// TIA Portal V20 program export: 2 tag tables, 2 data types, 5 data blocks, 11 code blocks (in call order from the OBs), 10 instance data blocks

VAR_GLOBAL   // PLC tag table "PLC_Centralizer_PLC_Production_And_Rework"
   In AT %I500.0 : "IO_Device_Inputs";
   Out AT %Q500.0 : "IO_Device_Outputs";
END_VAR

VAR_GLOBAL   // PLC tag table "PLC_Production_And_Rework"
   Emergency_Stop_Release AT %I0.0 : Bool;
   Sensor_Water_Fountain_Before_Entrace_Functional_Test_Spinner_Conveyor_Belt AT %I0.1 : Bool;
   Sensor_Water_Fountain_Entrace_Functional_Test_Spinner_Conveyor_Belt AT %I0.2 : Bool;
   Sensor_Water_Fountain_Entrace_Functional_Test_After_Spinner_Conveyor_Belt AT %I0.3 : Bool;
   Trigger_Read_Serial_Number_Entrace_Functional_Test AT %I0.4 : Bool;
   Sensor_Water_Fountain_Geting_Exit_Rework_Conveyor_Belt AT %I0.5 : Bool;
   Button_Water_Fountain_Get_Exit_Rework_Conveyor_Belt AT %I0.6 : Bool;
   Trigger_Read_Serial_Number_Exit_Functional_Test AT %I0.7 : Bool;
   Sensor_Water_Fountain_Exit_Functional_Test_Spinner_Conveyor_Belt AT %I1.0 : Bool;
   Sensor_Water_Fountain_Exit_Functional_Test_After_Spinner_Conveyor_Belt AT %I1.1 : Bool;
   Sensor_Water_Fountain_Geting_Entrace_Rework_Conveyor_Belt_Start AT %I1.2 : Bool;
   Sensor_Water_Fountain_Geting_Entrace_Rework_Conveyor_Belt_Finish AT %I1.3 : Bool;
   Carousel_Frequency_Inverter_Fail AT %I1.4 : Bool;
   Conveyor_Belt_Functional_Test_Inverter_Fail AT %I1.5 : Bool;
   Selected_Voltage_220V AT %I8.0 : Bool;
   Selected_Voltage_127V AT %I8.1 : Bool;
   Sensor_Spinner_Entrace_Functional_Test_Position_Withdrawn AT %I8.2 : Bool;
   Sensor_Spinner_Entrace_Functional_Test_Position_Advanced AT %I8.3 : Bool;
   Sensor_Spinner_Exit_Functional_Test_Position_Withdrawn AT %I8.4 : Bool;
   Sensor_Spinner_Exit_Functional_Test_Position_Advanced AT %I8.5 : Bool;
   Digital_Input_20 AT %I8.6 : Bool;
   Digital_Input_21 AT %I8.7 : Bool;
   Digital_Input_22 AT %I9.0 : Bool;
   Digital_Input_23 AT %I9.1 : Bool;
   Digital_Input_24 AT %I9.2 : Bool;
   Digital_Input_25 AT %I9.3 : Bool;
   Digital_Input_26 AT %I9.4 : Bool;
   Digital_Input_27 AT %I9.5 : Bool;
   Digital_Input_28 AT %I9.6 : Bool;
   Digital_Input_29 AT %I9.7 : Bool;
   Analogic_Input_0 AT %IW64 : Int;
   Analogic_Input_1 AT %IW66 : Int;
   Spin_Carousel_Frequency_Inverter_Speed_1 AT %Q0.0 : Bool;
   Spin_Carousel_Frequency_Inverter_Speed_2 AT %Q0.1 : Bool;
   Spin_Carousel_Frequency_Inverter_Speed_3 AT %Q0.2 : Bool;
   Conveyor_Belt_Frequency_Inverter_Speed_1 AT %Q0.3 : Bool;
   Conveyor_Belt_Frequency_Inverter_Speed_2 AT %Q0.4 : Bool;
   Conveyor_Belt_Frequency_Inverter_Speed_3 AT %Q0.5 : Bool;
   Turn_On_Conveyor_Belt_Motor_Spinner_Get_Entrace_Function_Test AT %Q0.6 : Bool;
   Turn_On_Conveyor_Belt_Motor_Rework_Conveyor_Belt_Get_Entrace_Functional_Test AT %Q0.7 : Bool;
   Turn_On_Conveyor_Belt_Motor_Spinner_Get_Exit_Functional_Test AT %Q1.0 : Bool;
   Turn_On_Conveyor_Belt_Motor_Rework_Conveyor_Belt_Get_Exit_Funcional_Test AT %Q1.1 : Bool;
   Open_Air_Pressure AT %Q8.0 : Bool;
   Valve_Advance_Spinner_Entrace_Functional_Test AT %Q8.1 : Bool;
   Valve_Advance_Spinner_Exit_Functional_Test AT %Q8.2 : Bool;
   Signal_Pre_Functional_Test_Production_Line AT %Q8.3 : Bool;
   Digital_Output_14 AT %Q8.4 : Bool;
   Digital_Output_15 AT %Q8.5 : Bool;
   Digital_Output_16 AT %Q8.6 : Bool;
   Digital_Output_17 AT %Q8.7 : Bool;
   Digital_Output_18 AT %Q9.0 : Bool;
   Digital_Output_19 AT %Q9.1 : Bool;
   Digital_Output_20 AT %Q9.2 : Bool;
   Digital_Output_21 AT %Q9.3 : Bool;
   Digital_Output_22 AT %Q9.4 : Bool;
   Digital_Output_23 AT %Q9.5 : Bool;
   Voltage_220V_Selected AT %Q9.6 : Bool;
   Voltage_127V_Selected AT %Q9.7 : Bool;
   Clock_Byte AT %MB0 : Byte;
   Clock_10Hz AT %M0.0 : Bool;
   Clock_5Hz AT %M0.1 : Bool;
   "Clock_2.5Hz" AT %M0.2 : Bool;
   Clock_2Hz AT %M0.3 : Bool;
   "Clock_1.25Hz" AT %M0.4 : Bool;
   Clock_1Hz AT %M0.5 : Bool;
   "Clock_0.625Hz" AT %M0.6 : Bool;
   "Clock_0.5Hz" AT %M0.7 : Bool;
   System_Byte AT %MB1 : Byte;
   FirstScan AT %M1.0 : Bool;
   DiagStatusUpdate AT %M1.1 : Bool;
   AlwaysTRUE AT %M1.2 : Bool;
   AlwaysFALSE AT %M1.3 : Bool;
END_VAR

TYPE "IO_Device_Inputs"
   STRUCT
      Start : Bool;
      Manual_Turn_On_Motor_Caroussel : Bool;
      Manual_Turn_On_Motor_Conveyor_Belt : Bool;
      Water_Foutain_Fail_Functional_Test : Bool;
      Select_Motor_Speed : SInt;
      Carousel_Voltage_Selection : SInt;
   END_STRUCT;
END_TYPE

TYPE "IO_Device_Outputs"
   STRUCT
      Life_Trigger : Bool;
      Emergency_Stop_Release : Bool;
      Trigger_Read_Serial_Number_Entrace_Functional_Test : Bool;
      Trigger_Read_Serial_Number_Exit_Functional_Test : Bool;
      Selected_Voltage_220V : Bool;
      Selected_Voltage_127V : Bool;
      Carousel_Frequency_Inverter_Fail : Bool;
      Conveyor_Belt_Functional_Test_Inverter_Fail : Bool;
   END_STRUCT;
END_TYPE

DATA_BLOCK "DB_Analogic_Input"   // DB2
{ S7_Optimized_Access := 'TRUE' }
// stored: MemoryReserve 100
   VAR
      Real_Analogic_Input_0 : Real;
      Real_Analogic_Input_1 : Real;
      UInt_Analogic_Input_0 : UInt;
      UInt_Analogic_Input_1 : UInt;
   END_VAR
BEGIN
END_DATA_BLOCK

DATA_BLOCK "DB_Contron_Coveyor_Belt"   // DB5
{ S7_Optimized_Access := 'TRUE' }
// stored: MemoryReserve 100
   VAR
      Pause_Conveyor_Belt_And_Carousel_Functional_Test : Bool;
   END_VAR
BEGIN
END_DATA_BLOCK

DATA_BLOCK "DB_Digital_Input"   // DB1
{ S7_Optimized_Access := 'TRUE' }
// stored: MemoryReserve 100
   VAR
      Emergency_Stop_Release : Bool;
      Sensor_Water_Fountain_Before_Entrace_Functional_Test_Spinner_Conveyor_Belt : Bool;
      Sensor_Water_Fountain_Entrace_Functional_Test_Spinner_Conveyor_Belt : Bool;
      Sensor_Water_Fountain_Entrace_Functional_Test_After_Spinner_Conveyor_Belt : Bool;
      Trigger_Read_Serial_Number_Entrace_Functional_Test : Bool;
      Sensor_Water_Fountain_Geting_Exit_Rework_Conveyor_Belt : Bool;
      Button_Water_Fountain_Get_Exit_Rework_Conveyor_Belt : Bool;
      Trigger_Read_Serial_Number_Exit_Functional_Test : Bool;
      Sensor_Water_Fountain_Exit_Functional_Test_Spinner_Conveyor_Belt : Bool;
      Sensor_Water_Fountain_Exit_Functional_Test_After_Spinner_Conveyor_Belt : Bool;
      Sensor_Water_Fountain_Geting_Entrace_Rework_Conveyor_Belt_Start : Bool;
      Sensor_Water_Fountain_Geting_Entrace_Rework_Conveyor_Belt_Finish : Bool;
      Carousel_Frequency_Inverter_Fail : Bool;
      Conveyor_Belt_Functional_Test_Inverter_Fail : Bool;
      Selected_Voltage_220V : Bool;
      Selected_Voltage_127V : Bool;
      Sensor_Spinner_Entrace_Functional_Test_Position_Withdrawn : Bool;
      Sensor_Spinner_Entrace_Functional_Test_Position_Advanced : Bool;
      Sensor_Spinner_Exit_Functional_Test_Position_Withdrawn : Bool;
      Sensor_Spinner_Exit_Functional_Test_Position_Advanced : Bool;
      Digital_Input_20 : Bool;
      Digital_Input_21 : Bool;
      Digital_Input_22 : Bool;
      Digital_Input_23 : Bool;
      Digital_Input_24 : Bool;
      Digital_Input_25 : Bool;
      Digital_Input_26 : Bool;
      Digital_Input_27 : Bool;
      Digital_Input_28 : Bool;
      Digital_Input_29 : Bool;
   END_VAR
BEGIN
END_DATA_BLOCK

DATA_BLOCK "DB_Digital_Output"   // DB3
{ S7_Optimized_Access := 'TRUE' }
// stored: AutoNumber false, MemoryReserve 100
   VAR
      Spin_Carousel_Frequency_Inverter_Speed_1 : Bool;
      Spin_Carousel_Frequency_Inverter_Speed_2 : Bool;
      Spin_Carousel_Frequency_Inverter_Speed_3 : Bool;
      Conveyor_Belt_Frequency_Inverter_Speed_1 : Bool;
      Conveyor_Belt_Frequency_Inverter_Speed_2 : Bool;
      Conveyor_Belt_Frequency_Inverter_Speed_3 : Bool;
      Turn_On_Conveyor_Belt_Motor_Spinner_Get_Entrace_Function_Test : Bool;
      Turn_On_Conveyor_Belt_Motor_Rework_Conveyor_Belt_Get_Entrace_Functional_Test : Bool;
      Turn_On_Conveyor_Belt_Motor_Spinner_Get_Exit_Functional_Test : Bool;
      Turn_On_Conveyor_Belt_Motor_Rework_Conveyor_Belt_Get_Exit_Funcional_Test : Bool;
      Open_Air_Pressure : Bool;
      Valve_Advance_Spinner_Entrace_Functional_Test : Bool;
      Valve_Advance_Spinner_Exit_Functional_Test : Bool;
      Signal_Pre_Functional_Test_Production_Line : Bool;
      Digital_Output_14 : Bool;
      Digital_Output_15 : Bool;
      Digital_Output_16 : Bool;
      Digital_Output_17 : Bool;
      Digital_Output_18 : Bool;
      Digital_Output_19 : Bool;
      Digital_Output_20 : Bool;
      Digital_Output_21 : Bool;
      Digital_Output_22 : Bool;
      Digital_Output_23 : Bool;
      Voltage_220V_Selected : Bool;
      Voltage_127V_Selected : Bool;
   END_VAR
BEGIN
END_DATA_BLOCK

DATA_BLOCK "DB_Info_From_PCL_Centralizer"   // DB4
{ S7_Optimized_Access := 'TRUE' }
// stored: MemoryReserve 100
   VAR
      Start : Bool;
      Manual_Turn_On_Motor_Caroussel : Bool;
      Manual_Turn_On_Motor_Conveyor_Belt : Bool;
      Water_Foutain_Fail_Functional_Test : Bool;
      Select_Motor_Speed : SInt;
      Carousel_Voltage_Selection : SInt;
   END_VAR
BEGIN
END_DATA_BLOCK

ORGANIZATION_BLOCK "Main"   // OB1, LAD, ProgramCycle
TITLE = "Main Program Sweep (Cycle)"
{ S7_Optimized_Access := 'TRUE' }
// stored: SetENOAutomatically false
   VAR_INPUT
      Initial_Call : Bool;   // Initial call of this OB
      Remanence : Bool;   // =True, if remanent data are available
   END_VAR
BEGIN

REGION Network 1
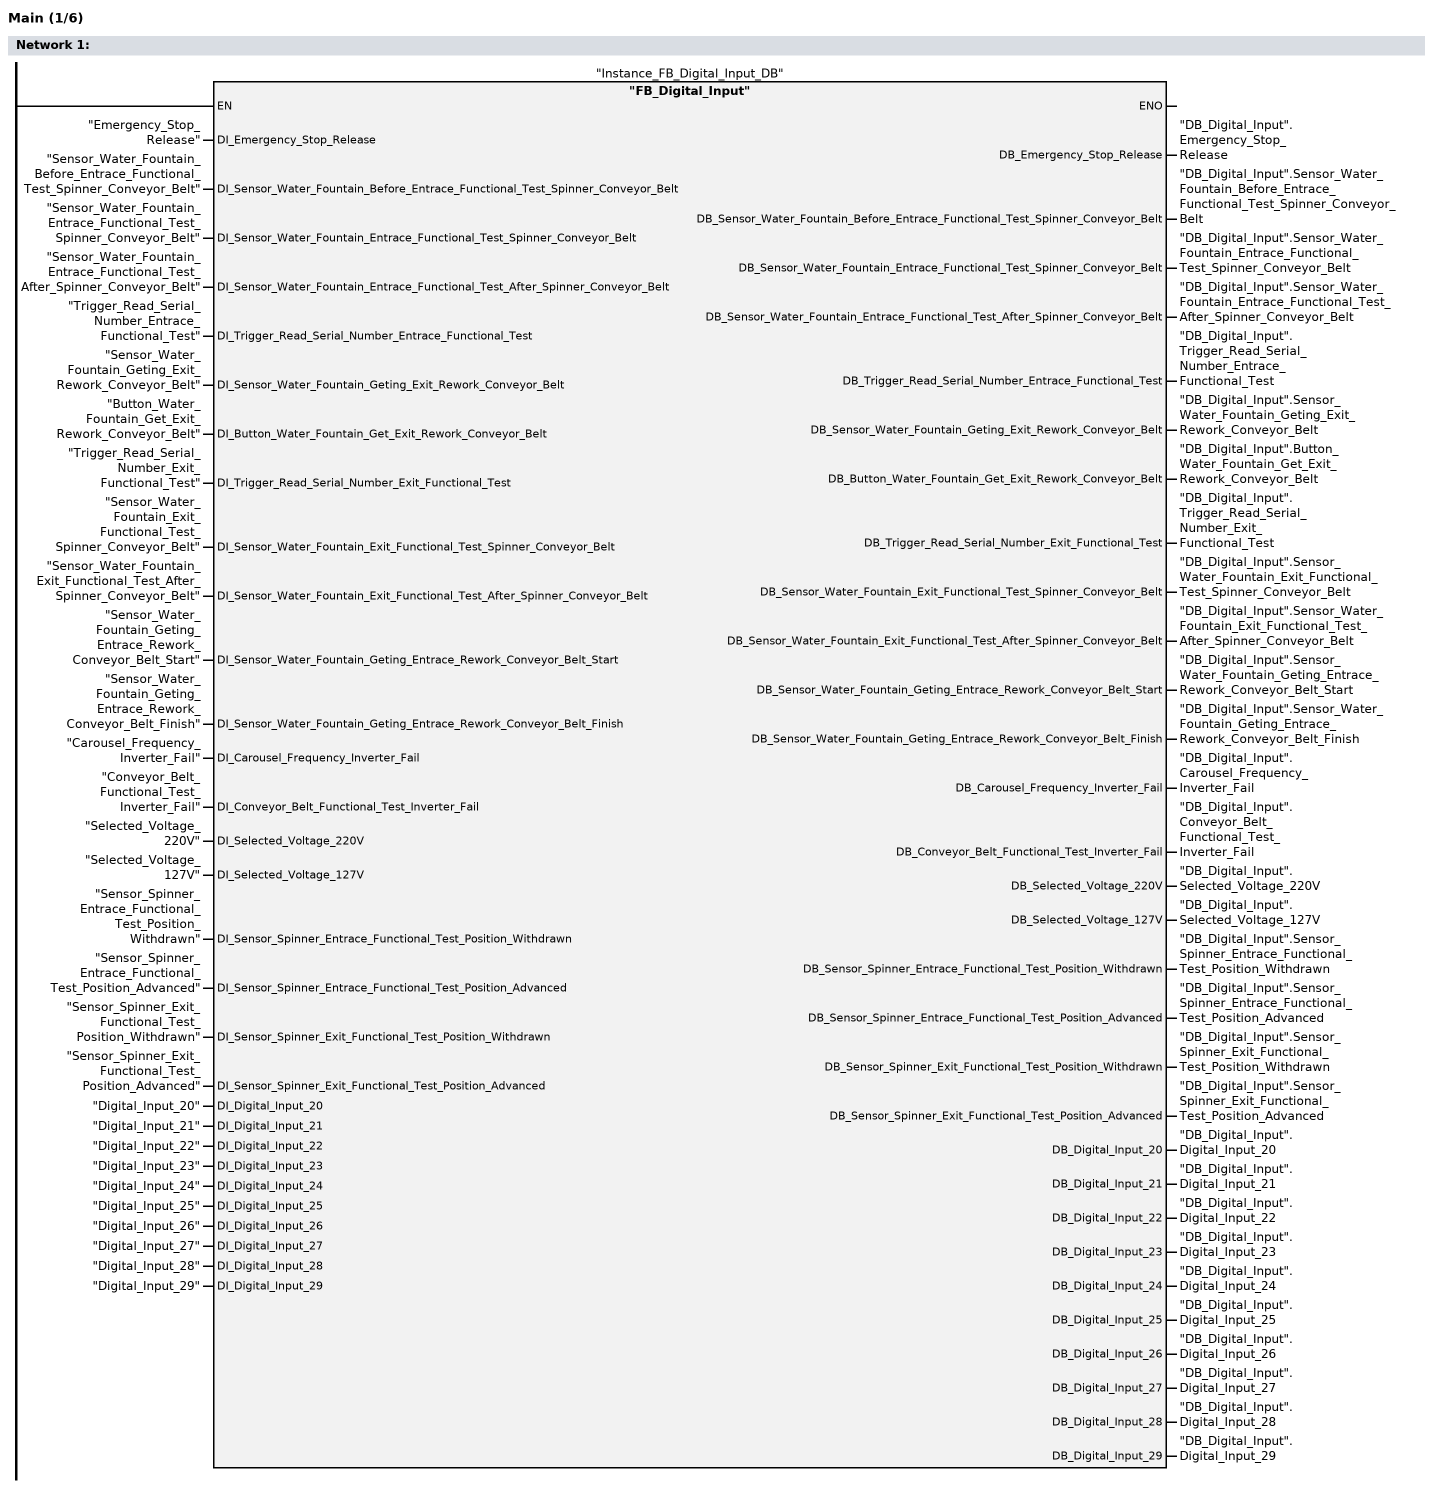
   RUNG wire#powerrail
      "Instance_FB_Digital_Input_DB"(DI_Emergency_Stop_Release := "Emergency_Stop_Release", DI_Sensor_Water_Fountain_Before_Entrace_Functional_Test_Spinner_Conveyor_Belt := "Sensor_Water_Fountain_Before_Entrace_Functional_Test_Spinner_Conveyor_Belt", DI_Sensor_Water_Fountain_Entrace_Functional_Test_Spinner_Conveyor_Belt := "Sensor_Water_Fountain_Entrace_Functional_Test_Spinner_Conveyor_Belt", DI_Sensor_Water_Fountain_Entrace_Functional_Test_After_Spinner_Conveyor_Belt := "Sensor_Water_Fountain_Entrace_Functional_Test_After_Spinner_Conveyor_Belt", DI_Trigger_Read_Serial_Number_Entrace_Functional_Test := "Trigger_Read_Serial_Number_Entrace_Functional_Test", DI_Sensor_Water_Fountain_Geting_Exit_Rework_Conveyor_Belt := "Sensor_Water_Fountain_Geting_Exit_Rework_Conveyor_Belt", DI_Button_Water_Fountain_Get_Exit_Rework_Conveyor_Belt := "Button_Water_Fountain_Get_Exit_Rework_Conveyor_Belt", DI_Trigger_Read_Serial_Number_Exit_Functional_Test := "Trigger_Read_Serial_Number_Exit_Functional_Test", DI_Sensor_Water_Fountain_Exit_Functional_Test_Spinner_Conveyor_Belt := "Sensor_Water_Fountain_Exit_Functional_Test_Spinner_Conveyor_Belt", DI_Sensor_Water_Fountain_Exit_Functional_Test_After_Spinner_Conveyor_Belt := "Sensor_Water_Fountain_Exit_Functional_Test_After_Spinner_Conveyor_Belt", DI_Sensor_Water_Fountain_Geting_Entrace_Rework_Conveyor_Belt_Start := "Sensor_Water_Fountain_Geting_Entrace_Rework_Conveyor_Belt_Start", DI_Sensor_Water_Fountain_Geting_Entrace_Rework_Conveyor_Belt_Finish := "Sensor_Water_Fountain_Geting_Entrace_Rework_Conveyor_Belt_Finish", DI_Carousel_Frequency_Inverter_Fail := "Carousel_Frequency_Inverter_Fail", DI_Conveyor_Belt_Functional_Test_Inverter_Fail := "Conveyor_Belt_Functional_Test_Inverter_Fail", DI_Selected_Voltage_220V := "Selected_Voltage_220V", DI_Selected_Voltage_127V := "Selected_Voltage_127V", DI_Sensor_Spinner_Entrace_Functional_Test_Position_Withdrawn := "Sensor_Spinner_Entrace_Functional_Test_Position_Withdrawn", DI_Sensor_Spinner_Entrace_Functional_Test_Position_Advanced := "Sensor_Spinner_Entrace_Functional_Test_Position_Advanced", DI_Sensor_Spinner_Exit_Functional_Test_Position_Withdrawn := "Sensor_Spinner_Exit_Functional_Test_Position_Withdrawn", DI_Sensor_Spinner_Exit_Functional_Test_Position_Advanced := "Sensor_Spinner_Exit_Functional_Test_Position_Advanced", DI_Digital_Input_20 := "Digital_Input_20", DI_Digital_Input_21 := "Digital_Input_21", DI_Digital_Input_22 := "Digital_Input_22", DI_Digital_Input_23 := "Digital_Input_23", DI_Digital_Input_24 := "Digital_Input_24", DI_Digital_Input_25 := "Digital_Input_25", DI_Digital_Input_26 := "Digital_Input_26", DI_Digital_Input_27 := "Digital_Input_27", DI_Digital_Input_28 := "Digital_Input_28", DI_Digital_Input_29 := "Digital_Input_29", DB_Emergency_Stop_Release => "DB_Digital_Input".Emergency_Stop_Release, DB_Sensor_Water_Fountain_Before_Entrace_Functional_Test_Spinner_Conveyor_Belt => "DB_Digital_Input".Sensor_Water_Fountain_Before_Entrace_Functional_Test_Spinner_Conveyor_Belt, DB_Sensor_Water_Fountain_Entrace_Functional_Test_Spinner_Conveyor_Belt => "DB_Digital_Input".Sensor_Water_Fountain_Entrace_Functional_Test_Spinner_Conveyor_Belt, DB_Sensor_Water_Fountain_Entrace_Functional_Test_After_Spinner_Conveyor_Belt => "DB_Digital_Input".Sensor_Water_Fountain_Entrace_Functional_Test_After_Spinner_Conveyor_Belt, DB_Trigger_Read_Serial_Number_Entrace_Functional_Test => "DB_Digital_Input".Trigger_Read_Serial_Number_Entrace_Functional_Test, DB_Sensor_Water_Fountain_Geting_Exit_Rework_Conveyor_Belt => "DB_Digital_Input".Sensor_Water_Fountain_Geting_Exit_Rework_Conveyor_Belt, DB_Button_Water_Fountain_Get_Exit_Rework_Conveyor_Belt => "DB_Digital_Input".Button_Water_Fountain_Get_Exit_Rework_Conveyor_Belt, DB_Trigger_Read_Serial_Number_Exit_Functional_Test => "DB_Digital_Input".Trigger_Read_Serial_Number_Exit_Functional_Test, DB_Sensor_Water_Fountain_Exit_Functional_Test_Spinner_Conveyor_Belt => "DB_Digital_Input".Sensor_Water_Fountain_Exit_Functional_Test_Spinner_Conveyor_Belt, DB_Sensor_Water_Fountain_Exit_Functional_Test_After_Spinner_Conveyor_Belt => "DB_Digital_Input".Sensor_Water_Fountain_Exit_Functional_Test_After_Spinner_Conveyor_Belt, DB_Sensor_Water_Fountain_Geting_Entrace_Rework_Conveyor_Belt_Start => "DB_Digital_Input".Sensor_Water_Fountain_Geting_Entrace_Rework_Conveyor_Belt_Start, DB_Sensor_Water_Fountain_Geting_Entrace_Rework_Conveyor_Belt_Finish => "DB_Digital_Input".Sensor_Water_Fountain_Geting_Entrace_Rework_Conveyor_Belt_Finish, DB_Carousel_Frequency_Inverter_Fail => "DB_Digital_Input".Carousel_Frequency_Inverter_Fail, DB_Conveyor_Belt_Functional_Test_Inverter_Fail => "DB_Digital_Input".Conveyor_Belt_Functional_Test_Inverter_Fail, DB_Selected_Voltage_220V => "DB_Digital_Input".Selected_Voltage_220V, DB_Selected_Voltage_127V => "DB_Digital_Input".Selected_Voltage_127V, DB_Sensor_Spinner_Entrace_Functional_Test_Position_Withdrawn => "DB_Digital_Input".Sensor_Spinner_Entrace_Functional_Test_Position_Withdrawn, DB_Sensor_Spinner_Entrace_Functional_Test_Position_Advanced => "DB_Digital_Input".Sensor_Spinner_Entrace_Functional_Test_Position_Advanced, DB_Sensor_Spinner_Exit_Functional_Test_Position_Withdrawn => "DB_Digital_Input".Sensor_Spinner_Exit_Functional_Test_Position_Withdrawn, DB_Sensor_Spinner_Exit_Functional_Test_Position_Advanced => "DB_Digital_Input".Sensor_Spinner_Exit_Functional_Test_Position_Advanced, DB_Digital_Input_20 => "DB_Digital_Input".Digital_Input_20, DB_Digital_Input_21 => "DB_Digital_Input".Digital_Input_21, DB_Digital_Input_22 => "DB_Digital_Input".Digital_Input_22, DB_Digital_Input_23 => "DB_Digital_Input".Digital_Input_23, DB_Digital_Input_24 => "DB_Digital_Input".Digital_Input_24, DB_Digital_Input_25 => "DB_Digital_Input".Digital_Input_25, DB_Digital_Input_26 => "DB_Digital_Input".Digital_Input_26, DB_Digital_Input_27 => "DB_Digital_Input".Digital_Input_27, DB_Digital_Input_28 => "DB_Digital_Input".Digital_Input_28, DB_Digital_Input_29 => "DB_Digital_Input".Digital_Input_29)
   END_RUNG
   // the same network as SCL:
   "Instance_FB_Digital_Input_DB"(DI_Emergency_Stop_Release := "Emergency_Stop_Release",   // "FB_Digital_Input"
                           DI_Sensor_Water_Fountain_Before_Entrace_Functional_Test_Spinner_Conveyor_Belt := "Sensor_Water_Fountain_Before_Entrace_Functional_Test_Spinner_Conveyor_Belt",
                           DI_Sensor_Water_Fountain_Entrace_Functional_Test_Spinner_Conveyor_Belt := "Sensor_Water_Fountain_Entrace_Functional_Test_Spinner_Conveyor_Belt",
                           DI_Sensor_Water_Fountain_Entrace_Functional_Test_After_Spinner_Conveyor_Belt := "Sensor_Water_Fountain_Entrace_Functional_Test_After_Spinner_Conveyor_Belt",
                           DI_Trigger_Read_Serial_Number_Entrace_Functional_Test := "Trigger_Read_Serial_Number_Entrace_Functional_Test",
                           DI_Sensor_Water_Fountain_Geting_Exit_Rework_Conveyor_Belt := "Sensor_Water_Fountain_Geting_Exit_Rework_Conveyor_Belt",
                           DI_Button_Water_Fountain_Get_Exit_Rework_Conveyor_Belt := "Button_Water_Fountain_Get_Exit_Rework_Conveyor_Belt",
                           DI_Trigger_Read_Serial_Number_Exit_Functional_Test := "Trigger_Read_Serial_Number_Exit_Functional_Test",
                           DI_Sensor_Water_Fountain_Exit_Functional_Test_Spinner_Conveyor_Belt := "Sensor_Water_Fountain_Exit_Functional_Test_Spinner_Conveyor_Belt",
                           DI_Sensor_Water_Fountain_Exit_Functional_Test_After_Spinner_Conveyor_Belt := "Sensor_Water_Fountain_Exit_Functional_Test_After_Spinner_Conveyor_Belt",
                           DI_Sensor_Water_Fountain_Geting_Entrace_Rework_Conveyor_Belt_Start := "Sensor_Water_Fountain_Geting_Entrace_Rework_Conveyor_Belt_Start",
                           DI_Sensor_Water_Fountain_Geting_Entrace_Rework_Conveyor_Belt_Finish := "Sensor_Water_Fountain_Geting_Entrace_Rework_Conveyor_Belt_Finish",
                           DI_Carousel_Frequency_Inverter_Fail := "Carousel_Frequency_Inverter_Fail",
                           DI_Conveyor_Belt_Functional_Test_Inverter_Fail := "Conveyor_Belt_Functional_Test_Inverter_Fail",
                           DI_Selected_Voltage_220V := "Selected_Voltage_220V",
                           DI_Selected_Voltage_127V := "Selected_Voltage_127V",
                           DI_Sensor_Spinner_Entrace_Functional_Test_Position_Withdrawn := "Sensor_Spinner_Entrace_Functional_Test_Position_Withdrawn",
                           DI_Sensor_Spinner_Entrace_Functional_Test_Position_Advanced := "Sensor_Spinner_Entrace_Functional_Test_Position_Advanced",
                           DI_Sensor_Spinner_Exit_Functional_Test_Position_Withdrawn := "Sensor_Spinner_Exit_Functional_Test_Position_Withdrawn",
                           DI_Sensor_Spinner_Exit_Functional_Test_Position_Advanced := "Sensor_Spinner_Exit_Functional_Test_Position_Advanced",
                           DI_Digital_Input_20 := "Digital_Input_20",
                           DI_Digital_Input_21 := "Digital_Input_21",
                           DI_Digital_Input_22 := "Digital_Input_22",
                           DI_Digital_Input_23 := "Digital_Input_23",
                           DI_Digital_Input_24 := "Digital_Input_24",
                           DI_Digital_Input_25 := "Digital_Input_25",
                           DI_Digital_Input_26 := "Digital_Input_26",
                           DI_Digital_Input_27 := "Digital_Input_27",
                           DI_Digital_Input_28 := "Digital_Input_28",
                           DI_Digital_Input_29 := "Digital_Input_29",
                           DB_Emergency_Stop_Release => "DB_Digital_Input".Emergency_Stop_Release,
                           DB_Sensor_Water_Fountain_Before_Entrace_Functional_Test_Spinner_Conveyor_Belt => "DB_Digital_Input".Sensor_Water_Fountain_Before_Entrace_Functional_Test_Spinner_Conveyor_Belt,
                           DB_Sensor_Water_Fountain_Entrace_Functional_Test_Spinner_Conveyor_Belt => "DB_Digital_Input".Sensor_Water_Fountain_Entrace_Functional_Test_Spinner_Conveyor_Belt,
                           DB_Sensor_Water_Fountain_Entrace_Functional_Test_After_Spinner_Conveyor_Belt => "DB_Digital_Input".Sensor_Water_Fountain_Entrace_Functional_Test_After_Spinner_Conveyor_Belt,
                           DB_Trigger_Read_Serial_Number_Entrace_Functional_Test => "DB_Digital_Input".Trigger_Read_Serial_Number_Entrace_Functional_Test,
                           DB_Sensor_Water_Fountain_Geting_Exit_Rework_Conveyor_Belt => "DB_Digital_Input".Sensor_Water_Fountain_Geting_Exit_Rework_Conveyor_Belt,
                           DB_Button_Water_Fountain_Get_Exit_Rework_Conveyor_Belt => "DB_Digital_Input".Button_Water_Fountain_Get_Exit_Rework_Conveyor_Belt,
                           DB_Trigger_Read_Serial_Number_Exit_Functional_Test => "DB_Digital_Input".Trigger_Read_Serial_Number_Exit_Functional_Test,
                           DB_Sensor_Water_Fountain_Exit_Functional_Test_Spinner_Conveyor_Belt => "DB_Digital_Input".Sensor_Water_Fountain_Exit_Functional_Test_Spinner_Conveyor_Belt,
                           DB_Sensor_Water_Fountain_Exit_Functional_Test_After_Spinner_Conveyor_Belt => "DB_Digital_Input".Sensor_Water_Fountain_Exit_Functional_Test_After_Spinner_Conveyor_Belt,
                           DB_Sensor_Water_Fountain_Geting_Entrace_Rework_Conveyor_Belt_Start => "DB_Digital_Input".Sensor_Water_Fountain_Geting_Entrace_Rework_Conveyor_Belt_Start,
                           DB_Sensor_Water_Fountain_Geting_Entrace_Rework_Conveyor_Belt_Finish => "DB_Digital_Input".Sensor_Water_Fountain_Geting_Entrace_Rework_Conveyor_Belt_Finish,
                           DB_Carousel_Frequency_Inverter_Fail => "DB_Digital_Input".Carousel_Frequency_Inverter_Fail,
                           DB_Conveyor_Belt_Functional_Test_Inverter_Fail => "DB_Digital_Input".Conveyor_Belt_Functional_Test_Inverter_Fail,
                           DB_Selected_Voltage_220V => "DB_Digital_Input".Selected_Voltage_220V,
                           DB_Selected_Voltage_127V => "DB_Digital_Input".Selected_Voltage_127V,
                           DB_Sensor_Spinner_Entrace_Functional_Test_Position_Withdrawn => "DB_Digital_Input".Sensor_Spinner_Entrace_Functional_Test_Position_Withdrawn,
                           DB_Sensor_Spinner_Entrace_Functional_Test_Position_Advanced => "DB_Digital_Input".Sensor_Spinner_Entrace_Functional_Test_Position_Advanced,
                           DB_Sensor_Spinner_Exit_Functional_Test_Position_Withdrawn => "DB_Digital_Input".Sensor_Spinner_Exit_Functional_Test_Position_Withdrawn,
                           DB_Sensor_Spinner_Exit_Functional_Test_Position_Advanced => "DB_Digital_Input".Sensor_Spinner_Exit_Functional_Test_Position_Advanced,
                           DB_Digital_Input_20 => "DB_Digital_Input".Digital_Input_20,
                           DB_Digital_Input_21 => "DB_Digital_Input".Digital_Input_21,
                           DB_Digital_Input_22 => "DB_Digital_Input".Digital_Input_22,
                           DB_Digital_Input_23 => "DB_Digital_Input".Digital_Input_23,
                           DB_Digital_Input_24 => "DB_Digital_Input".Digital_Input_24,
                           DB_Digital_Input_25 => "DB_Digital_Input".Digital_Input_25,
                           DB_Digital_Input_26 => "DB_Digital_Input".Digital_Input_26,
                           DB_Digital_Input_27 => "DB_Digital_Input".Digital_Input_27,
                           DB_Digital_Input_28 => "DB_Digital_Input".Digital_Input_28,
                           DB_Digital_Input_29 => "DB_Digital_Input".Digital_Input_29);
END_REGION

REGION Network 2
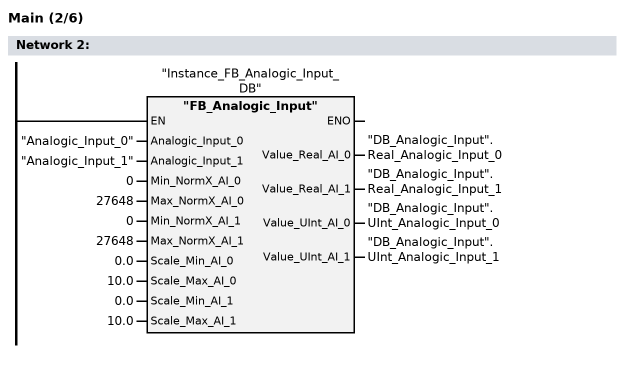
   RUNG wire#powerrail
      "Instance_FB_Analogic_Input_DB"(Analogic_Input_0 := "Analogic_Input_0", Analogic_Input_1 := "Analogic_Input_1", Min_NormX_AI_0 := 0, Max_NormX_AI_0 := 27648, Min_NormX_AI_1 := 0, Max_NormX_AI_1 := 27648, Scale_Min_AI_0 := 0.0, Scale_Max_AI_0 := 10.0, Scale_Min_AI_1 := 0.0, Scale_Max_AI_1 := 10.0, Value_Real_AI_0 => "DB_Analogic_Input".Real_Analogic_Input_0, Value_Real_AI_1 => "DB_Analogic_Input".Real_Analogic_Input_1, Value_UInt_AI_0 => "DB_Analogic_Input".UInt_Analogic_Input_0, Value_UInt_AI_1 => "DB_Analogic_Input".UInt_Analogic_Input_1)
   END_RUNG
   // the same network as SCL:
   "Instance_FB_Analogic_Input_DB"(Analogic_Input_0 := "Analogic_Input_0",   // "FB_Analogic_Input"
                           Analogic_Input_1 := "Analogic_Input_1",
                           Min_NormX_AI_0 := 0,
                           Max_NormX_AI_0 := 27648,
                           Min_NormX_AI_1 := 0,
                           Max_NormX_AI_1 := 27648,
                           Scale_Min_AI_0 := 0.0,
                           Scale_Max_AI_0 := 10.0,
                           Scale_Min_AI_1 := 0.0,
                           Scale_Max_AI_1 := 10.0,
                           Value_Real_AI_0 => "DB_Analogic_Input".Real_Analogic_Input_0,
                           Value_Real_AI_1 => "DB_Analogic_Input".Real_Analogic_Input_1,
                           Value_UInt_AI_0 => "DB_Analogic_Input".UInt_Analogic_Input_0,
                           Value_UInt_AI_1 => "DB_Analogic_Input".UInt_Analogic_Input_1);
END_REGION

REGION Network 3
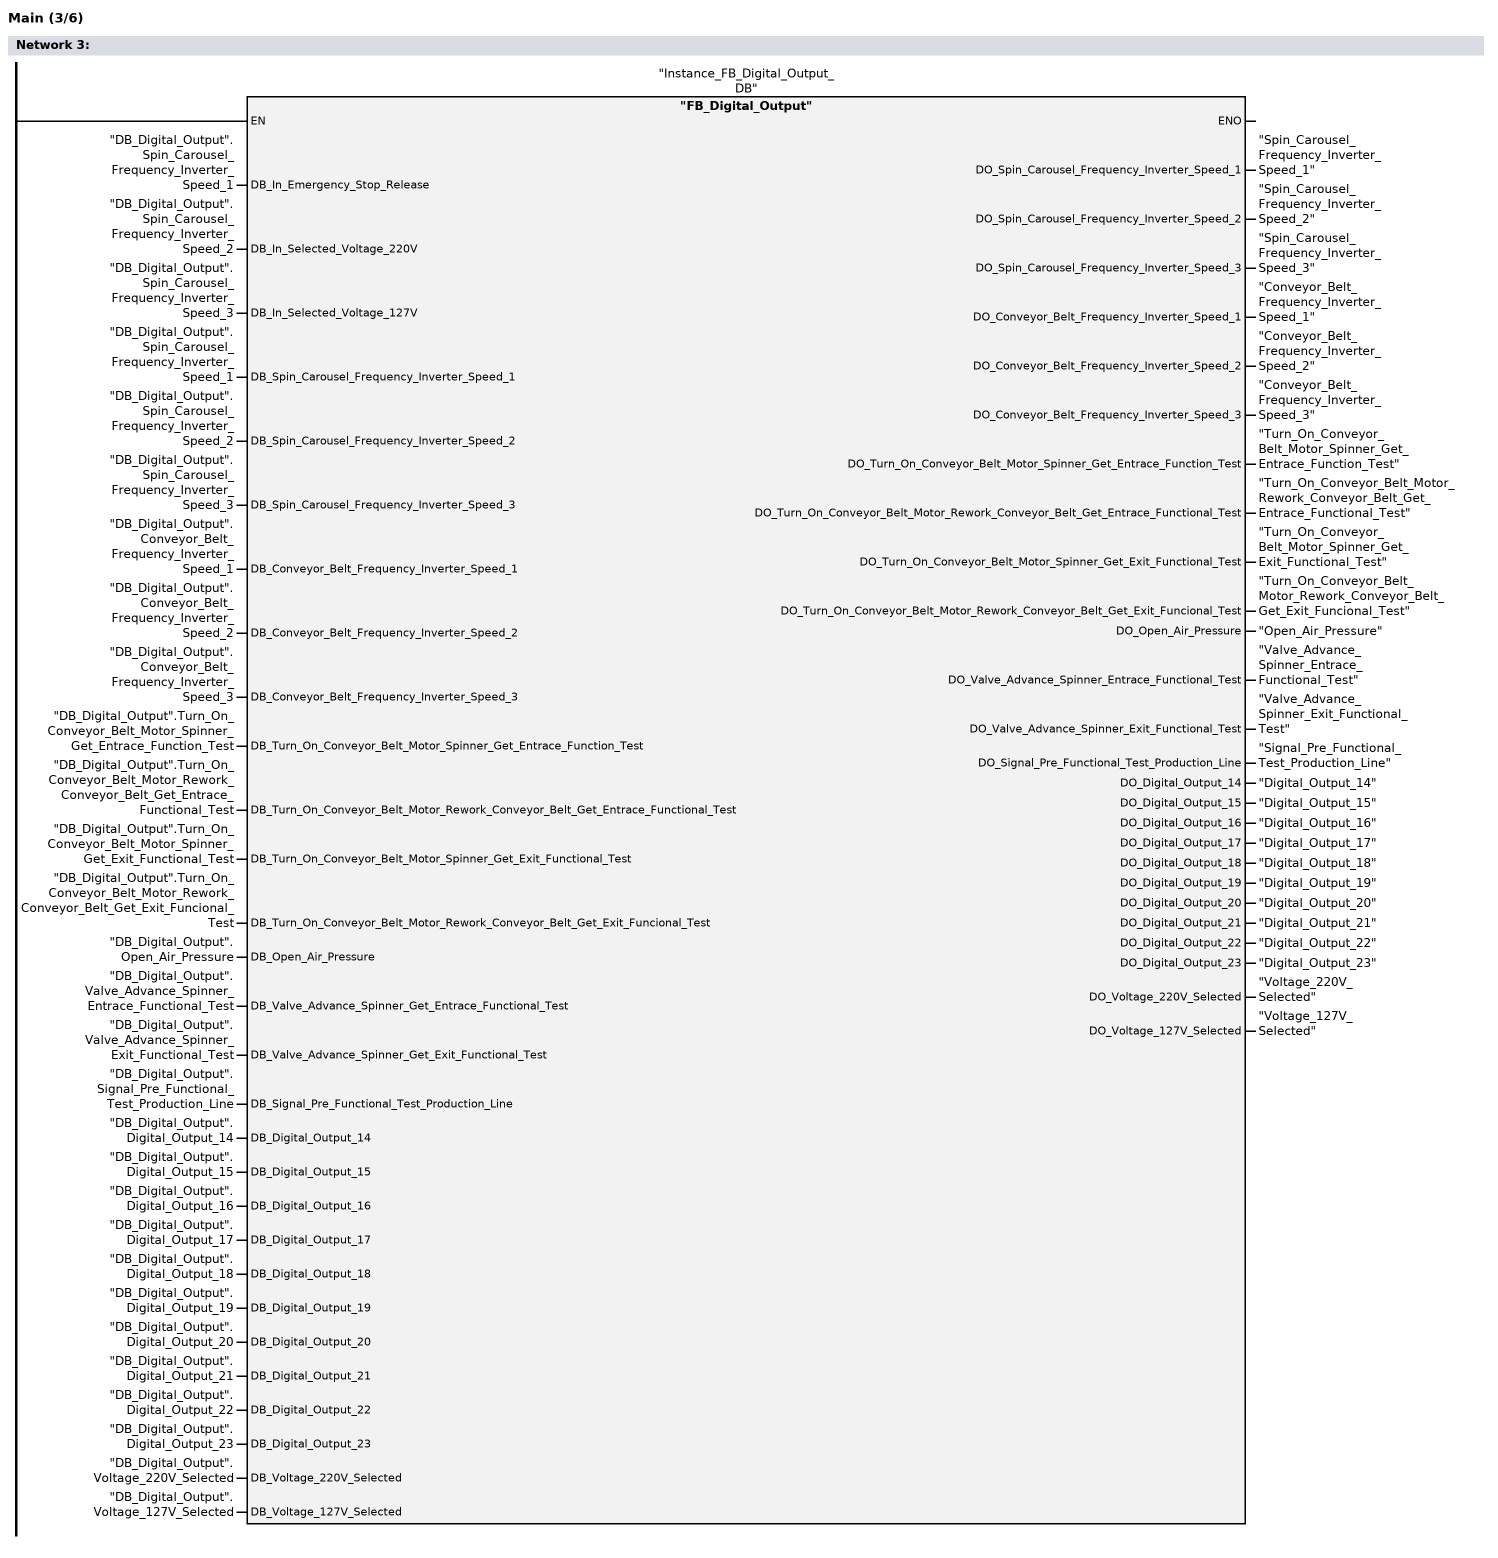
   RUNG wire#powerrail
      "Instance_FB_Digital_Output_DB"(DB_In_Emergency_Stop_Release := "DB_Digital_Output".Spin_Carousel_Frequency_Inverter_Speed_1, DB_In_Selected_Voltage_220V := "DB_Digital_Output".Spin_Carousel_Frequency_Inverter_Speed_2, DB_In_Selected_Voltage_127V := "DB_Digital_Output".Spin_Carousel_Frequency_Inverter_Speed_3, DB_Spin_Carousel_Frequency_Inverter_Speed_1 := "DB_Digital_Output".Spin_Carousel_Frequency_Inverter_Speed_1, DB_Spin_Carousel_Frequency_Inverter_Speed_2 := "DB_Digital_Output".Spin_Carousel_Frequency_Inverter_Speed_2, DB_Spin_Carousel_Frequency_Inverter_Speed_3 := "DB_Digital_Output".Spin_Carousel_Frequency_Inverter_Speed_3, DB_Conveyor_Belt_Frequency_Inverter_Speed_1 := "DB_Digital_Output".Conveyor_Belt_Frequency_Inverter_Speed_1, DB_Conveyor_Belt_Frequency_Inverter_Speed_2 := "DB_Digital_Output".Conveyor_Belt_Frequency_Inverter_Speed_2, DB_Conveyor_Belt_Frequency_Inverter_Speed_3 := "DB_Digital_Output".Conveyor_Belt_Frequency_Inverter_Speed_3, DB_Turn_On_Conveyor_Belt_Motor_Spinner_Get_Entrace_Function_Test := "DB_Digital_Output".Turn_On_Conveyor_Belt_Motor_Spinner_Get_Entrace_Function_Test, DB_Turn_On_Conveyor_Belt_Motor_Rework_Conveyor_Belt_Get_Entrace_Functional_Test := "DB_Digital_Output".Turn_On_Conveyor_Belt_Motor_Rework_Conveyor_Belt_Get_Entrace_Functional_Test, DB_Turn_On_Conveyor_Belt_Motor_Spinner_Get_Exit_Functional_Test := "DB_Digital_Output".Turn_On_Conveyor_Belt_Motor_Spinner_Get_Exit_Functional_Test, DB_Turn_On_Conveyor_Belt_Motor_Rework_Conveyor_Belt_Get_Exit_Funcional_Test := "DB_Digital_Output".Turn_On_Conveyor_Belt_Motor_Rework_Conveyor_Belt_Get_Exit_Funcional_Test, DB_Open_Air_Pressure := "DB_Digital_Output".Open_Air_Pressure, DB_Valve_Advance_Spinner_Get_Entrace_Functional_Test := "DB_Digital_Output".Valve_Advance_Spinner_Entrace_Functional_Test, DB_Valve_Advance_Spinner_Get_Exit_Functional_Test := "DB_Digital_Output".Valve_Advance_Spinner_Exit_Functional_Test, DB_Signal_Pre_Functional_Test_Production_Line := "DB_Digital_Output".Signal_Pre_Functional_Test_Production_Line, DB_Digital_Output_14 := "DB_Digital_Output".Digital_Output_14, DB_Digital_Output_15 := "DB_Digital_Output".Digital_Output_15, DB_Digital_Output_16 := "DB_Digital_Output".Digital_Output_16, DB_Digital_Output_17 := "DB_Digital_Output".Digital_Output_17, DB_Digital_Output_18 := "DB_Digital_Output".Digital_Output_18, DB_Digital_Output_19 := "DB_Digital_Output".Digital_Output_19, DB_Digital_Output_20 := "DB_Digital_Output".Digital_Output_20, DB_Digital_Output_21 := "DB_Digital_Output".Digital_Output_21, DB_Digital_Output_22 := "DB_Digital_Output".Digital_Output_22, DB_Digital_Output_23 := "DB_Digital_Output".Digital_Output_23, DB_Voltage_220V_Selected := "DB_Digital_Output".Voltage_220V_Selected, DB_Voltage_127V_Selected := "DB_Digital_Output".Voltage_127V_Selected, DO_Spin_Carousel_Frequency_Inverter_Speed_1 => "Spin_Carousel_Frequency_Inverter_Speed_1", DO_Spin_Carousel_Frequency_Inverter_Speed_2 => "Spin_Carousel_Frequency_Inverter_Speed_2", DO_Spin_Carousel_Frequency_Inverter_Speed_3 => "Spin_Carousel_Frequency_Inverter_Speed_3", DO_Conveyor_Belt_Frequency_Inverter_Speed_1 => "Conveyor_Belt_Frequency_Inverter_Speed_1", DO_Conveyor_Belt_Frequency_Inverter_Speed_2 => "Conveyor_Belt_Frequency_Inverter_Speed_2", DO_Conveyor_Belt_Frequency_Inverter_Speed_3 => "Conveyor_Belt_Frequency_Inverter_Speed_3", DO_Turn_On_Conveyor_Belt_Motor_Spinner_Get_Entrace_Function_Test => "Turn_On_Conveyor_Belt_Motor_Spinner_Get_Entrace_Function_Test", DO_Turn_On_Conveyor_Belt_Motor_Rework_Conveyor_Belt_Get_Entrace_Functional_Test => "Turn_On_Conveyor_Belt_Motor_Rework_Conveyor_Belt_Get_Entrace_Functional_Test", DO_Turn_On_Conveyor_Belt_Motor_Spinner_Get_Exit_Functional_Test => "Turn_On_Conveyor_Belt_Motor_Spinner_Get_Exit_Functional_Test", DO_Turn_On_Conveyor_Belt_Motor_Rework_Conveyor_Belt_Get_Exit_Funcional_Test => "Turn_On_Conveyor_Belt_Motor_Rework_Conveyor_Belt_Get_Exit_Funcional_Test", DO_Open_Air_Pressure => "Open_Air_Pressure", DO_Valve_Advance_Spinner_Entrace_Functional_Test => "Valve_Advance_Spinner_Entrace_Functional_Test", DO_Valve_Advance_Spinner_Exit_Functional_Test => "Valve_Advance_Spinner_Exit_Functional_Test", DO_Signal_Pre_Functional_Test_Production_Line => "Signal_Pre_Functional_Test_Production_Line", DO_Digital_Output_14 => "Digital_Output_14", DO_Digital_Output_15 => "Digital_Output_15", DO_Digital_Output_16 => "Digital_Output_16", DO_Digital_Output_17 => "Digital_Output_17", DO_Digital_Output_18 => "Digital_Output_18", DO_Digital_Output_19 => "Digital_Output_19", DO_Digital_Output_20 => "Digital_Output_20", DO_Digital_Output_21 => "Digital_Output_21", DO_Digital_Output_22 => "Digital_Output_22", DO_Digital_Output_23 => "Digital_Output_23", DO_Voltage_220V_Selected => "Voltage_220V_Selected", DO_Voltage_127V_Selected => "Voltage_127V_Selected")
   END_RUNG
   // the same network as SCL:
   "Instance_FB_Digital_Output_DB"(DB_In_Emergency_Stop_Release := "DB_Digital_Output".Spin_Carousel_Frequency_Inverter_Speed_1,   // "FB_Digital_Output"
                           DB_In_Selected_Voltage_220V := "DB_Digital_Output".Spin_Carousel_Frequency_Inverter_Speed_2,
                           DB_In_Selected_Voltage_127V := "DB_Digital_Output".Spin_Carousel_Frequency_Inverter_Speed_3,
                           DB_Spin_Carousel_Frequency_Inverter_Speed_1 := "DB_Digital_Output".Spin_Carousel_Frequency_Inverter_Speed_1,
                           DB_Spin_Carousel_Frequency_Inverter_Speed_2 := "DB_Digital_Output".Spin_Carousel_Frequency_Inverter_Speed_2,
                           DB_Spin_Carousel_Frequency_Inverter_Speed_3 := "DB_Digital_Output".Spin_Carousel_Frequency_Inverter_Speed_3,
                           DB_Conveyor_Belt_Frequency_Inverter_Speed_1 := "DB_Digital_Output".Conveyor_Belt_Frequency_Inverter_Speed_1,
                           DB_Conveyor_Belt_Frequency_Inverter_Speed_2 := "DB_Digital_Output".Conveyor_Belt_Frequency_Inverter_Speed_2,
                           DB_Conveyor_Belt_Frequency_Inverter_Speed_3 := "DB_Digital_Output".Conveyor_Belt_Frequency_Inverter_Speed_3,
                           DB_Turn_On_Conveyor_Belt_Motor_Spinner_Get_Entrace_Function_Test := "DB_Digital_Output".Turn_On_Conveyor_Belt_Motor_Spinner_Get_Entrace_Function_Test,
                           DB_Turn_On_Conveyor_Belt_Motor_Rework_Conveyor_Belt_Get_Entrace_Functional_Test := "DB_Digital_Output".Turn_On_Conveyor_Belt_Motor_Rework_Conveyor_Belt_Get_Entrace_Functional_Test,
                           DB_Turn_On_Conveyor_Belt_Motor_Spinner_Get_Exit_Functional_Test := "DB_Digital_Output".Turn_On_Conveyor_Belt_Motor_Spinner_Get_Exit_Functional_Test,
                           DB_Turn_On_Conveyor_Belt_Motor_Rework_Conveyor_Belt_Get_Exit_Funcional_Test := "DB_Digital_Output".Turn_On_Conveyor_Belt_Motor_Rework_Conveyor_Belt_Get_Exit_Funcional_Test,
                           DB_Open_Air_Pressure := "DB_Digital_Output".Open_Air_Pressure,
                           DB_Valve_Advance_Spinner_Get_Entrace_Functional_Test := "DB_Digital_Output".Valve_Advance_Spinner_Entrace_Functional_Test,
                           DB_Valve_Advance_Spinner_Get_Exit_Functional_Test := "DB_Digital_Output".Valve_Advance_Spinner_Exit_Functional_Test,
                           DB_Signal_Pre_Functional_Test_Production_Line := "DB_Digital_Output".Signal_Pre_Functional_Test_Production_Line,
                           DB_Digital_Output_14 := "DB_Digital_Output".Digital_Output_14,
                           DB_Digital_Output_15 := "DB_Digital_Output".Digital_Output_15,
                           DB_Digital_Output_16 := "DB_Digital_Output".Digital_Output_16,
                           DB_Digital_Output_17 := "DB_Digital_Output".Digital_Output_17,
                           DB_Digital_Output_18 := "DB_Digital_Output".Digital_Output_18,
                           DB_Digital_Output_19 := "DB_Digital_Output".Digital_Output_19,
                           DB_Digital_Output_20 := "DB_Digital_Output".Digital_Output_20,
                           DB_Digital_Output_21 := "DB_Digital_Output".Digital_Output_21,
                           DB_Digital_Output_22 := "DB_Digital_Output".Digital_Output_22,
                           DB_Digital_Output_23 := "DB_Digital_Output".Digital_Output_23,
                           DB_Voltage_220V_Selected := "DB_Digital_Output".Voltage_220V_Selected,
                           DB_Voltage_127V_Selected := "DB_Digital_Output".Voltage_127V_Selected,
                           DO_Spin_Carousel_Frequency_Inverter_Speed_1 => "Spin_Carousel_Frequency_Inverter_Speed_1",
                           DO_Spin_Carousel_Frequency_Inverter_Speed_2 => "Spin_Carousel_Frequency_Inverter_Speed_2",
                           DO_Spin_Carousel_Frequency_Inverter_Speed_3 => "Spin_Carousel_Frequency_Inverter_Speed_3",
                           DO_Conveyor_Belt_Frequency_Inverter_Speed_1 => "Conveyor_Belt_Frequency_Inverter_Speed_1",
                           DO_Conveyor_Belt_Frequency_Inverter_Speed_2 => "Conveyor_Belt_Frequency_Inverter_Speed_2",
                           DO_Conveyor_Belt_Frequency_Inverter_Speed_3 => "Conveyor_Belt_Frequency_Inverter_Speed_3",
                           DO_Turn_On_Conveyor_Belt_Motor_Spinner_Get_Entrace_Function_Test => "Turn_On_Conveyor_Belt_Motor_Spinner_Get_Entrace_Function_Test",
                           DO_Turn_On_Conveyor_Belt_Motor_Rework_Conveyor_Belt_Get_Entrace_Functional_Test => "Turn_On_Conveyor_Belt_Motor_Rework_Conveyor_Belt_Get_Entrace_Functional_Test",
                           DO_Turn_On_Conveyor_Belt_Motor_Spinner_Get_Exit_Functional_Test => "Turn_On_Conveyor_Belt_Motor_Spinner_Get_Exit_Functional_Test",
                           DO_Turn_On_Conveyor_Belt_Motor_Rework_Conveyor_Belt_Get_Exit_Funcional_Test => "Turn_On_Conveyor_Belt_Motor_Rework_Conveyor_Belt_Get_Exit_Funcional_Test",
                           DO_Open_Air_Pressure => "Open_Air_Pressure",
                           DO_Valve_Advance_Spinner_Entrace_Functional_Test => "Valve_Advance_Spinner_Entrace_Functional_Test",
                           DO_Valve_Advance_Spinner_Exit_Functional_Test => "Valve_Advance_Spinner_Exit_Functional_Test",
                           DO_Signal_Pre_Functional_Test_Production_Line => "Signal_Pre_Functional_Test_Production_Line",
                           DO_Digital_Output_14 => "Digital_Output_14",
                           DO_Digital_Output_15 => "Digital_Output_15",
                           DO_Digital_Output_16 => "Digital_Output_16",
                           DO_Digital_Output_17 => "Digital_Output_17",
                           DO_Digital_Output_18 => "Digital_Output_18",
                           DO_Digital_Output_19 => "Digital_Output_19",
                           DO_Digital_Output_20 => "Digital_Output_20",
                           DO_Digital_Output_21 => "Digital_Output_21",
                           DO_Digital_Output_22 => "Digital_Output_22",
                           DO_Digital_Output_23 => "Digital_Output_23",
                           DO_Voltage_220V_Selected => "Voltage_220V_Selected",
                           DO_Voltage_127V_Selected => "Voltage_127V_Selected");
END_REGION

REGION Network 4
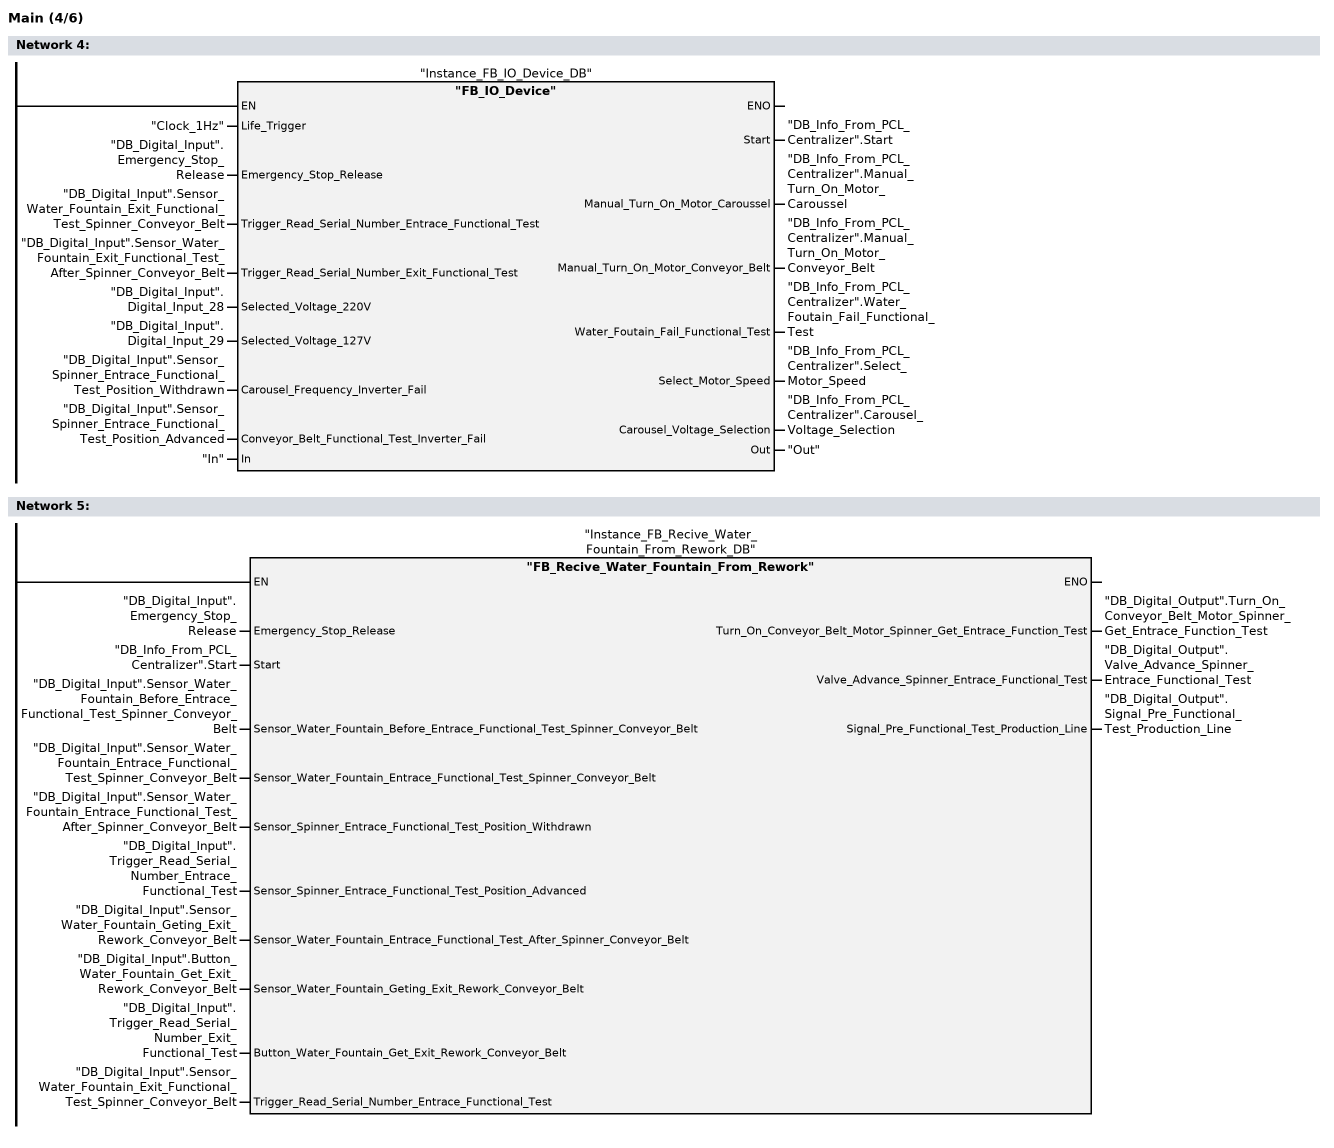
   RUNG wire#powerrail
      "Instance_FB_IO_Device_DB"(Life_Trigger := "Clock_1Hz", Emergency_Stop_Release := "DB_Digital_Input".Emergency_Stop_Release, Trigger_Read_Serial_Number_Entrace_Functional_Test := "DB_Digital_Input".Sensor_Water_Fountain_Exit_Functional_Test_Spinner_Conveyor_Belt, Trigger_Read_Serial_Number_Exit_Functional_Test := "DB_Digital_Input".Sensor_Water_Fountain_Exit_Functional_Test_After_Spinner_Conveyor_Belt, Selected_Voltage_220V := "DB_Digital_Input".Digital_Input_28, Selected_Voltage_127V := "DB_Digital_Input".Digital_Input_29, Carousel_Frequency_Inverter_Fail := "DB_Digital_Input".Sensor_Spinner_Entrace_Functional_Test_Position_Withdrawn, Conveyor_Belt_Functional_Test_Inverter_Fail := "DB_Digital_Input".Sensor_Spinner_Entrace_Functional_Test_Position_Advanced, In := "In", Start => "DB_Info_From_PCL_Centralizer".Start, Manual_Turn_On_Motor_Caroussel => "DB_Info_From_PCL_Centralizer".Manual_Turn_On_Motor_Caroussel, Manual_Turn_On_Motor_Conveyor_Belt => "DB_Info_From_PCL_Centralizer".Manual_Turn_On_Motor_Conveyor_Belt, Water_Foutain_Fail_Functional_Test => "DB_Info_From_PCL_Centralizer".Water_Foutain_Fail_Functional_Test, Select_Motor_Speed => "DB_Info_From_PCL_Centralizer".Select_Motor_Speed, Carousel_Voltage_Selection => "DB_Info_From_PCL_Centralizer".Carousel_Voltage_Selection, Out => "Out")
   END_RUNG
   // the same network as SCL:
   "Instance_FB_IO_Device_DB"(Life_Trigger := "Clock_1Hz",   // "FB_IO_Device"
                           Emergency_Stop_Release := "DB_Digital_Input".Emergency_Stop_Release,
                           Trigger_Read_Serial_Number_Entrace_Functional_Test := "DB_Digital_Input".Sensor_Water_Fountain_Exit_Functional_Test_Spinner_Conveyor_Belt,
                           Trigger_Read_Serial_Number_Exit_Functional_Test := "DB_Digital_Input".Sensor_Water_Fountain_Exit_Functional_Test_After_Spinner_Conveyor_Belt,
                           Selected_Voltage_220V := "DB_Digital_Input".Digital_Input_28,
                           Selected_Voltage_127V := "DB_Digital_Input".Digital_Input_29,
                           Carousel_Frequency_Inverter_Fail := "DB_Digital_Input".Sensor_Spinner_Entrace_Functional_Test_Position_Withdrawn,
                           Conveyor_Belt_Functional_Test_Inverter_Fail := "DB_Digital_Input".Sensor_Spinner_Entrace_Functional_Test_Position_Advanced,
                           In := "In",
                           Start => "DB_Info_From_PCL_Centralizer".Start,
                           Manual_Turn_On_Motor_Caroussel => "DB_Info_From_PCL_Centralizer".Manual_Turn_On_Motor_Caroussel,
                           Manual_Turn_On_Motor_Conveyor_Belt => "DB_Info_From_PCL_Centralizer".Manual_Turn_On_Motor_Conveyor_Belt,
                           Water_Foutain_Fail_Functional_Test => "DB_Info_From_PCL_Centralizer".Water_Foutain_Fail_Functional_Test,
                           Select_Motor_Speed => "DB_Info_From_PCL_Centralizer".Select_Motor_Speed,
                           Carousel_Voltage_Selection => "DB_Info_From_PCL_Centralizer".Carousel_Voltage_Selection,
                           Out => "Out");
END_REGION

REGION Network 5
   RUNG wire#powerrail
      "Instance_FB_Recive_Water_Fountain_From_Rework_DB"(Emergency_Stop_Release := "DB_Digital_Input".Emergency_Stop_Release, Start := "DB_Info_From_PCL_Centralizer".Start, Sensor_Water_Fountain_Before_Entrace_Functional_Test_Spinner_Conveyor_Belt := "DB_Digital_Input".Sensor_Water_Fountain_Before_Entrace_Functional_Test_Spinner_Conveyor_Belt, Sensor_Water_Fountain_Entrace_Functional_Test_Spinner_Conveyor_Belt := "DB_Digital_Input".Sensor_Water_Fountain_Entrace_Functional_Test_Spinner_Conveyor_Belt, Sensor_Spinner_Entrace_Functional_Test_Position_Withdrawn := "DB_Digital_Input".Sensor_Water_Fountain_Entrace_Functional_Test_After_Spinner_Conveyor_Belt, Sensor_Spinner_Entrace_Functional_Test_Position_Advanced := "DB_Digital_Input".Trigger_Read_Serial_Number_Entrace_Functional_Test, Sensor_Water_Fountain_Entrace_Functional_Test_After_Spinner_Conveyor_Belt := "DB_Digital_Input".Sensor_Water_Fountain_Geting_Exit_Rework_Conveyor_Belt, Sensor_Water_Fountain_Geting_Exit_Rework_Conveyor_Belt := "DB_Digital_Input".Button_Water_Fountain_Get_Exit_Rework_Conveyor_Belt, Button_Water_Fountain_Get_Exit_Rework_Conveyor_Belt := "DB_Digital_Input".Trigger_Read_Serial_Number_Exit_Functional_Test, Trigger_Read_Serial_Number_Entrace_Functional_Test := "DB_Digital_Input".Sensor_Water_Fountain_Exit_Functional_Test_Spinner_Conveyor_Belt, Turn_On_Conveyor_Belt_Motor_Spinner_Get_Entrace_Function_Test => "DB_Digital_Output".Turn_On_Conveyor_Belt_Motor_Spinner_Get_Entrace_Function_Test, Valve_Advance_Spinner_Entrace_Functional_Test => "DB_Digital_Output".Valve_Advance_Spinner_Entrace_Functional_Test, Signal_Pre_Functional_Test_Production_Line => "DB_Digital_Output".Signal_Pre_Functional_Test_Production_Line)
   END_RUNG
   // the same network as SCL:
   "Instance_FB_Recive_Water_Fountain_From_Rework_DB"(Emergency_Stop_Release := "DB_Digital_Input".Emergency_Stop_Release,   // "FB_Recive_Water_Fountain_From_Rework"
                           Start := "DB_Info_From_PCL_Centralizer".Start,
                           Sensor_Water_Fountain_Before_Entrace_Functional_Test_Spinner_Conveyor_Belt := "DB_Digital_Input".Sensor_Water_Fountain_Before_Entrace_Functional_Test_Spinner_Conveyor_Belt,
                           Sensor_Water_Fountain_Entrace_Functional_Test_Spinner_Conveyor_Belt := "DB_Digital_Input".Sensor_Water_Fountain_Entrace_Functional_Test_Spinner_Conveyor_Belt,
                           Sensor_Spinner_Entrace_Functional_Test_Position_Withdrawn := "DB_Digital_Input".Sensor_Water_Fountain_Entrace_Functional_Test_After_Spinner_Conveyor_Belt,
                           Sensor_Spinner_Entrace_Functional_Test_Position_Advanced := "DB_Digital_Input".Trigger_Read_Serial_Number_Entrace_Functional_Test,
                           Sensor_Water_Fountain_Entrace_Functional_Test_After_Spinner_Conveyor_Belt := "DB_Digital_Input".Sensor_Water_Fountain_Geting_Exit_Rework_Conveyor_Belt,
                           Sensor_Water_Fountain_Geting_Exit_Rework_Conveyor_Belt := "DB_Digital_Input".Button_Water_Fountain_Get_Exit_Rework_Conveyor_Belt,
                           Button_Water_Fountain_Get_Exit_Rework_Conveyor_Belt := "DB_Digital_Input".Trigger_Read_Serial_Number_Exit_Functional_Test,
                           Trigger_Read_Serial_Number_Entrace_Functional_Test := "DB_Digital_Input".Sensor_Water_Fountain_Exit_Functional_Test_Spinner_Conveyor_Belt,
                           Turn_On_Conveyor_Belt_Motor_Spinner_Get_Entrace_Function_Test => "DB_Digital_Output".Turn_On_Conveyor_Belt_Motor_Spinner_Get_Entrace_Function_Test,
                           Valve_Advance_Spinner_Entrace_Functional_Test => "DB_Digital_Output".Valve_Advance_Spinner_Entrace_Functional_Test,
                           Signal_Pre_Functional_Test_Production_Line => "DB_Digital_Output".Signal_Pre_Functional_Test_Production_Line);
END_REGION

REGION Network 6
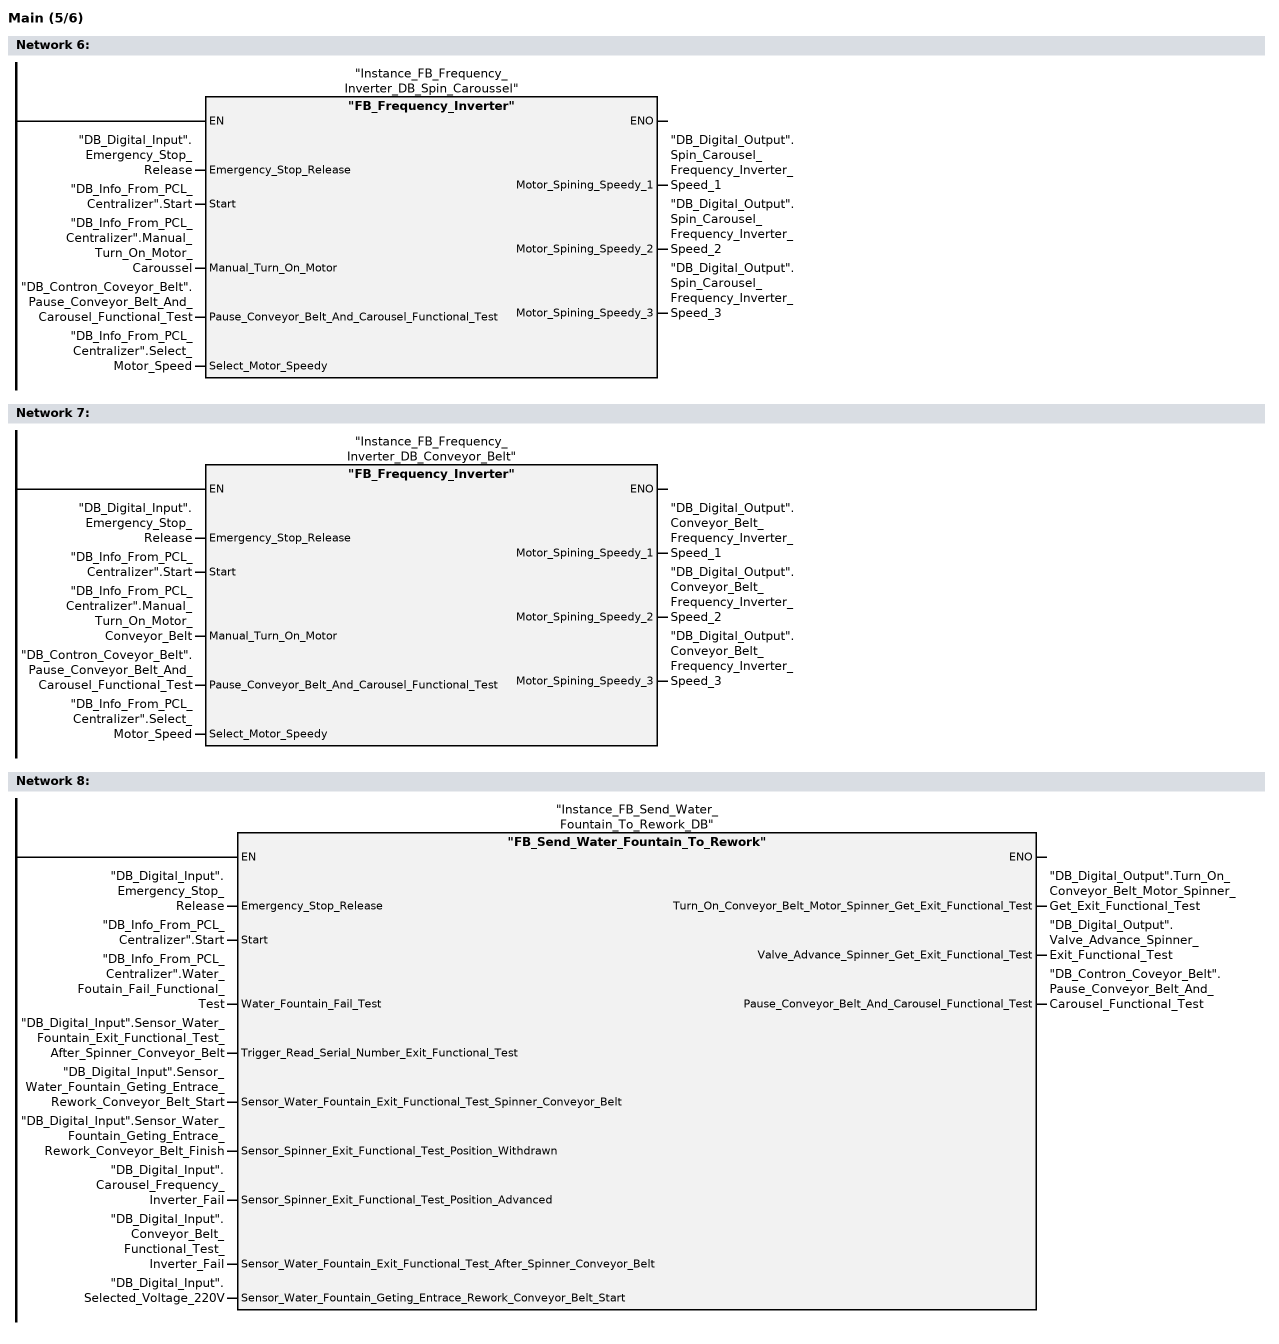
   RUNG wire#powerrail
      "Instance_FB_Frequency_Inverter_DB_Spin_Caroussel"(Emergency_Stop_Release := "DB_Digital_Input".Emergency_Stop_Release, Start := "DB_Info_From_PCL_Centralizer".Start, Manual_Turn_On_Motor := "DB_Info_From_PCL_Centralizer".Manual_Turn_On_Motor_Caroussel, Pause_Conveyor_Belt_And_Carousel_Functional_Test := "DB_Contron_Coveyor_Belt".Pause_Conveyor_Belt_And_Carousel_Functional_Test, Select_Motor_Speedy := "DB_Info_From_PCL_Centralizer".Select_Motor_Speed, Motor_Spining_Speedy_1 => "DB_Digital_Output".Spin_Carousel_Frequency_Inverter_Speed_1, Motor_Spining_Speedy_2 => "DB_Digital_Output".Spin_Carousel_Frequency_Inverter_Speed_2, Motor_Spining_Speedy_3 => "DB_Digital_Output".Spin_Carousel_Frequency_Inverter_Speed_3)
   END_RUNG
   // the same network as SCL:
   "Instance_FB_Frequency_Inverter_DB_Spin_Caroussel"(Emergency_Stop_Release := "DB_Digital_Input".Emergency_Stop_Release,   // "FB_Frequency_Inverter"
                           Start := "DB_Info_From_PCL_Centralizer".Start,
                           Manual_Turn_On_Motor := "DB_Info_From_PCL_Centralizer".Manual_Turn_On_Motor_Caroussel,
                           Pause_Conveyor_Belt_And_Carousel_Functional_Test := "DB_Contron_Coveyor_Belt".Pause_Conveyor_Belt_And_Carousel_Functional_Test,
                           Select_Motor_Speedy := "DB_Info_From_PCL_Centralizer".Select_Motor_Speed,
                           Motor_Spining_Speedy_1 => "DB_Digital_Output".Spin_Carousel_Frequency_Inverter_Speed_1,
                           Motor_Spining_Speedy_2 => "DB_Digital_Output".Spin_Carousel_Frequency_Inverter_Speed_2,
                           Motor_Spining_Speedy_3 => "DB_Digital_Output".Spin_Carousel_Frequency_Inverter_Speed_3);
END_REGION

REGION Network 7
   RUNG wire#powerrail
      "Instance_FB_Frequency_Inverter_DB_Conveyor_Belt"(Emergency_Stop_Release := "DB_Digital_Input".Emergency_Stop_Release, Start := "DB_Info_From_PCL_Centralizer".Start, Manual_Turn_On_Motor := "DB_Info_From_PCL_Centralizer".Manual_Turn_On_Motor_Conveyor_Belt, Pause_Conveyor_Belt_And_Carousel_Functional_Test := "DB_Contron_Coveyor_Belt".Pause_Conveyor_Belt_And_Carousel_Functional_Test, Select_Motor_Speedy := "DB_Info_From_PCL_Centralizer".Select_Motor_Speed, Motor_Spining_Speedy_1 => "DB_Digital_Output".Conveyor_Belt_Frequency_Inverter_Speed_1, Motor_Spining_Speedy_2 => "DB_Digital_Output".Conveyor_Belt_Frequency_Inverter_Speed_2, Motor_Spining_Speedy_3 => "DB_Digital_Output".Conveyor_Belt_Frequency_Inverter_Speed_3)
   END_RUNG
   // the same network as SCL:
   "Instance_FB_Frequency_Inverter_DB_Conveyor_Belt"(Emergency_Stop_Release := "DB_Digital_Input".Emergency_Stop_Release,   // "FB_Frequency_Inverter"
                           Start := "DB_Info_From_PCL_Centralizer".Start,
                           Manual_Turn_On_Motor := "DB_Info_From_PCL_Centralizer".Manual_Turn_On_Motor_Conveyor_Belt,
                           Pause_Conveyor_Belt_And_Carousel_Functional_Test := "DB_Contron_Coveyor_Belt".Pause_Conveyor_Belt_And_Carousel_Functional_Test,
                           Select_Motor_Speedy := "DB_Info_From_PCL_Centralizer".Select_Motor_Speed,
                           Motor_Spining_Speedy_1 => "DB_Digital_Output".Conveyor_Belt_Frequency_Inverter_Speed_1,
                           Motor_Spining_Speedy_2 => "DB_Digital_Output".Conveyor_Belt_Frequency_Inverter_Speed_2,
                           Motor_Spining_Speedy_3 => "DB_Digital_Output".Conveyor_Belt_Frequency_Inverter_Speed_3);
END_REGION

REGION Network 8
   RUNG wire#powerrail
      "Instance_FB_Send_Water_Fountain_To_Rework_DB"(Emergency_Stop_Release := "DB_Digital_Input".Emergency_Stop_Release, Start := "DB_Info_From_PCL_Centralizer".Start, Water_Fountain_Fail_Test := "DB_Info_From_PCL_Centralizer".Water_Foutain_Fail_Functional_Test, Trigger_Read_Serial_Number_Exit_Functional_Test := "DB_Digital_Input".Sensor_Water_Fountain_Exit_Functional_Test_After_Spinner_Conveyor_Belt, Sensor_Water_Fountain_Exit_Functional_Test_Spinner_Conveyor_Belt := "DB_Digital_Input".Sensor_Water_Fountain_Geting_Entrace_Rework_Conveyor_Belt_Start, Sensor_Spinner_Exit_Functional_Test_Position_Withdrawn := "DB_Digital_Input".Sensor_Water_Fountain_Geting_Entrace_Rework_Conveyor_Belt_Finish, Sensor_Spinner_Exit_Functional_Test_Position_Advanced := "DB_Digital_Input".Carousel_Frequency_Inverter_Fail, Sensor_Water_Fountain_Exit_Functional_Test_After_Spinner_Conveyor_Belt := "DB_Digital_Input".Conveyor_Belt_Functional_Test_Inverter_Fail, Sensor_Water_Fountain_Geting_Entrace_Rework_Conveyor_Belt_Start := "DB_Digital_Input".Selected_Voltage_220V, Turn_On_Conveyor_Belt_Motor_Spinner_Get_Exit_Functional_Test => "DB_Digital_Output".Turn_On_Conveyor_Belt_Motor_Spinner_Get_Exit_Functional_Test, Valve_Advance_Spinner_Get_Exit_Functional_Test => "DB_Digital_Output".Valve_Advance_Spinner_Exit_Functional_Test, Pause_Conveyor_Belt_And_Carousel_Functional_Test => "DB_Contron_Coveyor_Belt".Pause_Conveyor_Belt_And_Carousel_Functional_Test)
   END_RUNG
   // the same network as SCL:
   "Instance_FB_Send_Water_Fountain_To_Rework_DB"(Emergency_Stop_Release := "DB_Digital_Input".Emergency_Stop_Release,   // "FB_Send_Water_Fountain_To_Rework"
                           Start := "DB_Info_From_PCL_Centralizer".Start,
                           Water_Fountain_Fail_Test := "DB_Info_From_PCL_Centralizer".Water_Foutain_Fail_Functional_Test,
                           Trigger_Read_Serial_Number_Exit_Functional_Test := "DB_Digital_Input".Sensor_Water_Fountain_Exit_Functional_Test_After_Spinner_Conveyor_Belt,
                           Sensor_Water_Fountain_Exit_Functional_Test_Spinner_Conveyor_Belt := "DB_Digital_Input".Sensor_Water_Fountain_Geting_Entrace_Rework_Conveyor_Belt_Start,
                           Sensor_Spinner_Exit_Functional_Test_Position_Withdrawn := "DB_Digital_Input".Sensor_Water_Fountain_Geting_Entrace_Rework_Conveyor_Belt_Finish,
                           Sensor_Spinner_Exit_Functional_Test_Position_Advanced := "DB_Digital_Input".Carousel_Frequency_Inverter_Fail,
                           Sensor_Water_Fountain_Exit_Functional_Test_After_Spinner_Conveyor_Belt := "DB_Digital_Input".Conveyor_Belt_Functional_Test_Inverter_Fail,
                           Sensor_Water_Fountain_Geting_Entrace_Rework_Conveyor_Belt_Start := "DB_Digital_Input".Selected_Voltage_220V,
                           Turn_On_Conveyor_Belt_Motor_Spinner_Get_Exit_Functional_Test => "DB_Digital_Output".Turn_On_Conveyor_Belt_Motor_Spinner_Get_Exit_Functional_Test,
                           Valve_Advance_Spinner_Get_Exit_Functional_Test => "DB_Digital_Output".Valve_Advance_Spinner_Exit_Functional_Test,
                           Pause_Conveyor_Belt_And_Carousel_Functional_Test => "DB_Contron_Coveyor_Belt".Pause_Conveyor_Belt_And_Carousel_Functional_Test);
END_REGION

REGION Network 9
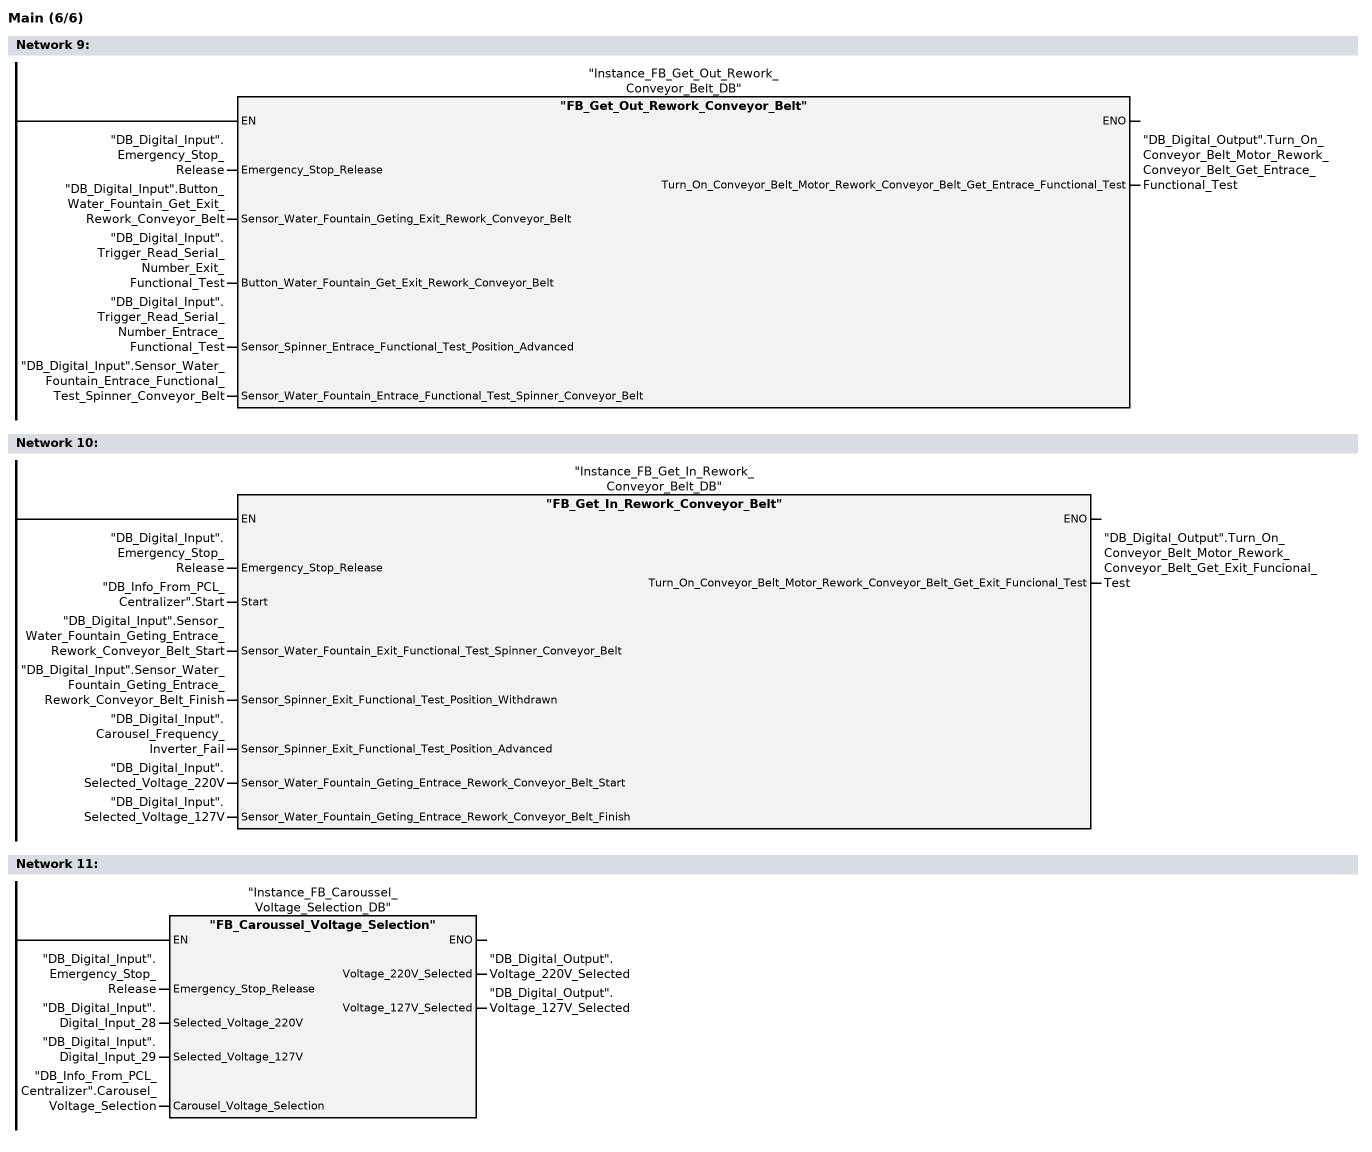
   RUNG wire#powerrail
      "Instance_FB_Get_Out_Rework_Conveyor_Belt_DB"(Emergency_Stop_Release := "DB_Digital_Input".Emergency_Stop_Release, Sensor_Water_Fountain_Geting_Exit_Rework_Conveyor_Belt := "DB_Digital_Input".Button_Water_Fountain_Get_Exit_Rework_Conveyor_Belt, Button_Water_Fountain_Get_Exit_Rework_Conveyor_Belt := "DB_Digital_Input".Trigger_Read_Serial_Number_Exit_Functional_Test, Sensor_Spinner_Entrace_Functional_Test_Position_Advanced := "DB_Digital_Input".Trigger_Read_Serial_Number_Entrace_Functional_Test, Sensor_Water_Fountain_Entrace_Functional_Test_Spinner_Conveyor_Belt := "DB_Digital_Input".Sensor_Water_Fountain_Entrace_Functional_Test_Spinner_Conveyor_Belt, Turn_On_Conveyor_Belt_Motor_Rework_Conveyor_Belt_Get_Entrace_Functional_Test => "DB_Digital_Output".Turn_On_Conveyor_Belt_Motor_Rework_Conveyor_Belt_Get_Entrace_Functional_Test)
   END_RUNG
   // the same network as SCL:
   "Instance_FB_Get_Out_Rework_Conveyor_Belt_DB"(Emergency_Stop_Release := "DB_Digital_Input".Emergency_Stop_Release,   // "FB_Get_Out_Rework_Conveyor_Belt"
                           Sensor_Water_Fountain_Geting_Exit_Rework_Conveyor_Belt := "DB_Digital_Input".Button_Water_Fountain_Get_Exit_Rework_Conveyor_Belt,
                           Button_Water_Fountain_Get_Exit_Rework_Conveyor_Belt := "DB_Digital_Input".Trigger_Read_Serial_Number_Exit_Functional_Test,
                           Sensor_Spinner_Entrace_Functional_Test_Position_Advanced := "DB_Digital_Input".Trigger_Read_Serial_Number_Entrace_Functional_Test,
                           Sensor_Water_Fountain_Entrace_Functional_Test_Spinner_Conveyor_Belt := "DB_Digital_Input".Sensor_Water_Fountain_Entrace_Functional_Test_Spinner_Conveyor_Belt,
                           Turn_On_Conveyor_Belt_Motor_Rework_Conveyor_Belt_Get_Entrace_Functional_Test => "DB_Digital_Output".Turn_On_Conveyor_Belt_Motor_Rework_Conveyor_Belt_Get_Entrace_Functional_Test);
END_REGION

REGION Network 10
   RUNG wire#powerrail
      "Instance_FB_Get_In_Rework_Conveyor_Belt_DB"(Emergency_Stop_Release := "DB_Digital_Input".Emergency_Stop_Release, Start := "DB_Info_From_PCL_Centralizer".Start, Sensor_Water_Fountain_Exit_Functional_Test_Spinner_Conveyor_Belt := "DB_Digital_Input".Sensor_Water_Fountain_Geting_Entrace_Rework_Conveyor_Belt_Start, Sensor_Spinner_Exit_Functional_Test_Position_Withdrawn := "DB_Digital_Input".Sensor_Water_Fountain_Geting_Entrace_Rework_Conveyor_Belt_Finish, Sensor_Spinner_Exit_Functional_Test_Position_Advanced := "DB_Digital_Input".Carousel_Frequency_Inverter_Fail, Sensor_Water_Fountain_Geting_Entrace_Rework_Conveyor_Belt_Start := "DB_Digital_Input".Selected_Voltage_220V, Sensor_Water_Fountain_Geting_Entrace_Rework_Conveyor_Belt_Finish := "DB_Digital_Input".Selected_Voltage_127V, Turn_On_Conveyor_Belt_Motor_Rework_Conveyor_Belt_Get_Exit_Funcional_Test => "DB_Digital_Output".Turn_On_Conveyor_Belt_Motor_Rework_Conveyor_Belt_Get_Exit_Funcional_Test)
   END_RUNG
   // the same network as SCL:
   "Instance_FB_Get_In_Rework_Conveyor_Belt_DB"(Emergency_Stop_Release := "DB_Digital_Input".Emergency_Stop_Release,   // "FB_Get_In_Rework_Conveyor_Belt"
                           Start := "DB_Info_From_PCL_Centralizer".Start,
                           Sensor_Water_Fountain_Exit_Functional_Test_Spinner_Conveyor_Belt := "DB_Digital_Input".Sensor_Water_Fountain_Geting_Entrace_Rework_Conveyor_Belt_Start,
                           Sensor_Spinner_Exit_Functional_Test_Position_Withdrawn := "DB_Digital_Input".Sensor_Water_Fountain_Geting_Entrace_Rework_Conveyor_Belt_Finish,
                           Sensor_Spinner_Exit_Functional_Test_Position_Advanced := "DB_Digital_Input".Carousel_Frequency_Inverter_Fail,
                           Sensor_Water_Fountain_Geting_Entrace_Rework_Conveyor_Belt_Start := "DB_Digital_Input".Selected_Voltage_220V,
                           Sensor_Water_Fountain_Geting_Entrace_Rework_Conveyor_Belt_Finish := "DB_Digital_Input".Selected_Voltage_127V,
                           Turn_On_Conveyor_Belt_Motor_Rework_Conveyor_Belt_Get_Exit_Funcional_Test => "DB_Digital_Output".Turn_On_Conveyor_Belt_Motor_Rework_Conveyor_Belt_Get_Exit_Funcional_Test);
END_REGION

REGION Network 11
   RUNG wire#powerrail
      "Instance_FB_Caroussel_Voltage_Selection_DB"(Emergency_Stop_Release := "DB_Digital_Input".Emergency_Stop_Release, Selected_Voltage_220V := "DB_Digital_Input".Digital_Input_28, Selected_Voltage_127V := "DB_Digital_Input".Digital_Input_29, Carousel_Voltage_Selection := "DB_Info_From_PCL_Centralizer".Carousel_Voltage_Selection, Voltage_220V_Selected => "DB_Digital_Output".Voltage_220V_Selected, Voltage_127V_Selected => "DB_Digital_Output".Voltage_127V_Selected)
   END_RUNG
   // the same network as SCL:
   "Instance_FB_Caroussel_Voltage_Selection_DB"(Emergency_Stop_Release := "DB_Digital_Input".Emergency_Stop_Release,   // "FB_Caroussel_Voltage_Selection"
                           Selected_Voltage_220V := "DB_Digital_Input".Digital_Input_28,
                           Selected_Voltage_127V := "DB_Digital_Input".Digital_Input_29,
                           Carousel_Voltage_Selection := "DB_Info_From_PCL_Centralizer".Carousel_Voltage_Selection,
                           Voltage_220V_Selected => "DB_Digital_Output".Voltage_220V_Selected,
                           Voltage_127V_Selected => "DB_Digital_Output".Voltage_127V_Selected);
END_REGION
END_ORGANIZATION_BLOCK

FUNCTION_BLOCK "FB_Digital_Input"   // FB1, LAD
{ S7_Optimized_Access := 'TRUE' }
// stored: MemoryReserve 100, SetENOAutomatically false
   VAR_INPUT
      DI_Emergency_Stop_Release : Bool;
      DI_Sensor_Water_Fountain_Before_Entrace_Functional_Test_Spinner_Conveyor_Belt : Bool;
      DI_Sensor_Water_Fountain_Entrace_Functional_Test_Spinner_Conveyor_Belt : Bool;
      DI_Sensor_Water_Fountain_Entrace_Functional_Test_After_Spinner_Conveyor_Belt : Bool;
      DI_Trigger_Read_Serial_Number_Entrace_Functional_Test : Bool;
      DI_Sensor_Water_Fountain_Geting_Exit_Rework_Conveyor_Belt : Bool;
      DI_Button_Water_Fountain_Get_Exit_Rework_Conveyor_Belt : Bool;
      DI_Trigger_Read_Serial_Number_Exit_Functional_Test : Bool;
      DI_Sensor_Water_Fountain_Exit_Functional_Test_Spinner_Conveyor_Belt : Bool;
      DI_Sensor_Water_Fountain_Exit_Functional_Test_After_Spinner_Conveyor_Belt : Bool;
      DI_Sensor_Water_Fountain_Geting_Entrace_Rework_Conveyor_Belt_Start : Bool;
      DI_Sensor_Water_Fountain_Geting_Entrace_Rework_Conveyor_Belt_Finish : Bool;
      DI_Carousel_Frequency_Inverter_Fail : Bool;
      DI_Conveyor_Belt_Functional_Test_Inverter_Fail : Bool;
      DI_Selected_Voltage_220V : Bool;
      DI_Selected_Voltage_127V : Bool;
      DI_Sensor_Spinner_Entrace_Functional_Test_Position_Withdrawn : Bool;
      DI_Sensor_Spinner_Entrace_Functional_Test_Position_Advanced : Bool;
      DI_Sensor_Spinner_Exit_Functional_Test_Position_Withdrawn : Bool;
      DI_Sensor_Spinner_Exit_Functional_Test_Position_Advanced : Bool;
      DI_Digital_Input_20 : Bool;
      DI_Digital_Input_21 : Bool;
      DI_Digital_Input_22 : Bool;
      DI_Digital_Input_23 : Bool;
      DI_Digital_Input_24 : Bool;
      DI_Digital_Input_25 : Bool;
      DI_Digital_Input_26 : Bool;
      DI_Digital_Input_27 : Bool;
      DI_Digital_Input_28 : Bool;
      DI_Digital_Input_29 : Bool;
   END_VAR
   VAR_OUTPUT
      DB_Emergency_Stop_Release : Bool;
      DB_Sensor_Water_Fountain_Before_Entrace_Functional_Test_Spinner_Conveyor_Belt : Bool;
      DB_Sensor_Water_Fountain_Entrace_Functional_Test_Spinner_Conveyor_Belt : Bool;
      DB_Sensor_Water_Fountain_Entrace_Functional_Test_After_Spinner_Conveyor_Belt : Bool;
      DB_Trigger_Read_Serial_Number_Entrace_Functional_Test : Bool;
      DB_Sensor_Water_Fountain_Geting_Exit_Rework_Conveyor_Belt : Bool;
      DB_Button_Water_Fountain_Get_Exit_Rework_Conveyor_Belt : Bool;
      DB_Trigger_Read_Serial_Number_Exit_Functional_Test : Bool;
      DB_Sensor_Water_Fountain_Exit_Functional_Test_Spinner_Conveyor_Belt : Bool;
      DB_Sensor_Water_Fountain_Exit_Functional_Test_After_Spinner_Conveyor_Belt : Bool;
      DB_Sensor_Water_Fountain_Geting_Entrace_Rework_Conveyor_Belt_Start : Bool;
      DB_Sensor_Water_Fountain_Geting_Entrace_Rework_Conveyor_Belt_Finish : Bool;
      DB_Carousel_Frequency_Inverter_Fail : Bool;
      DB_Conveyor_Belt_Functional_Test_Inverter_Fail : Bool;
      DB_Selected_Voltage_220V : Bool;
      DB_Selected_Voltage_127V : Bool;
      DB_Sensor_Spinner_Entrace_Functional_Test_Position_Withdrawn : Bool;
      DB_Sensor_Spinner_Entrace_Functional_Test_Position_Advanced : Bool;
      DB_Sensor_Spinner_Exit_Functional_Test_Position_Withdrawn : Bool;
      DB_Sensor_Spinner_Exit_Functional_Test_Position_Advanced : Bool;
      DB_Digital_Input_20 : Bool;
      DB_Digital_Input_21 : Bool;
      DB_Digital_Input_22 : Bool;
      DB_Digital_Input_23 : Bool;
      DB_Digital_Input_24 : Bool;
      DB_Digital_Input_25 : Bool;
      DB_Digital_Input_26 : Bool;
      DB_Digital_Input_27 : Bool;
      DB_Digital_Input_28 : Bool;
      DB_Digital_Input_29 : Bool;
   END_VAR
BEGIN

REGION Network 1
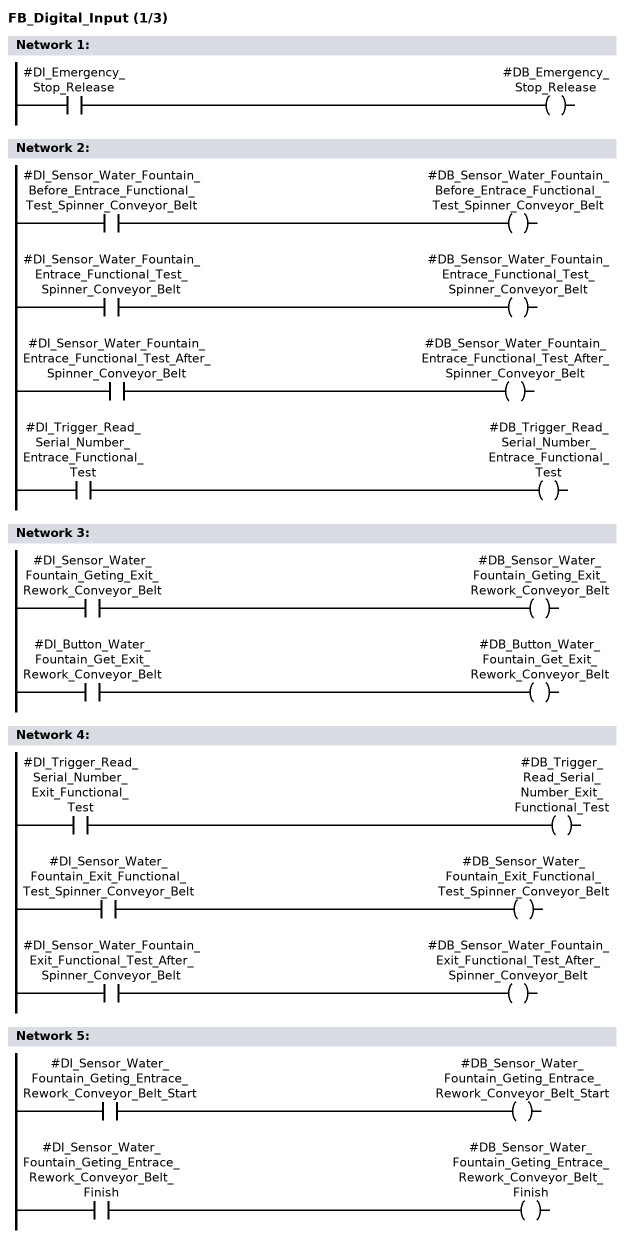
   RUNG wire#powerrail
      Contact( #DI_Emergency_Stop_Release )
      Coil( #DB_Emergency_Stop_Release )
   END_RUNG
   // the same network as SCL:
   #DB_Emergency_Stop_Release := #DI_Emergency_Stop_Release;
END_REGION

REGION Network 2
   RUNG wire#powerrail
      Contact( #DI_Sensor_Water_Fountain_Before_Entrace_Functional_Test_Spinner_Conveyor_Belt )
      Coil( #DB_Sensor_Water_Fountain_Before_Entrace_Functional_Test_Spinner_Conveyor_Belt )
   END_RUNG
   RUNG wire#powerrail
      Contact( #DI_Sensor_Water_Fountain_Entrace_Functional_Test_Spinner_Conveyor_Belt )
      Coil( #DB_Sensor_Water_Fountain_Entrace_Functional_Test_Spinner_Conveyor_Belt )
   END_RUNG
   RUNG wire#powerrail
      Contact( #DI_Sensor_Water_Fountain_Entrace_Functional_Test_After_Spinner_Conveyor_Belt )
      Coil( #DB_Sensor_Water_Fountain_Entrace_Functional_Test_After_Spinner_Conveyor_Belt )
   END_RUNG
   RUNG wire#powerrail
      Contact( #DI_Trigger_Read_Serial_Number_Entrace_Functional_Test )
      Coil( #DB_Trigger_Read_Serial_Number_Entrace_Functional_Test )
   END_RUNG
   // the same network as SCL:
   #DB_Sensor_Water_Fountain_Before_Entrace_Functional_Test_Spinner_Conveyor_Belt := #DI_Sensor_Water_Fountain_Before_Entrace_Functional_Test_Spinner_Conveyor_Belt;
   #DB_Sensor_Water_Fountain_Entrace_Functional_Test_Spinner_Conveyor_Belt := #DI_Sensor_Water_Fountain_Entrace_Functional_Test_Spinner_Conveyor_Belt;
   #DB_Sensor_Water_Fountain_Entrace_Functional_Test_After_Spinner_Conveyor_Belt := #DI_Sensor_Water_Fountain_Entrace_Functional_Test_After_Spinner_Conveyor_Belt;
   #DB_Trigger_Read_Serial_Number_Entrace_Functional_Test := #DI_Trigger_Read_Serial_Number_Entrace_Functional_Test;
END_REGION

REGION Network 3
   RUNG wire#powerrail
      Contact( #DI_Sensor_Water_Fountain_Geting_Exit_Rework_Conveyor_Belt )
      Coil( #DB_Sensor_Water_Fountain_Geting_Exit_Rework_Conveyor_Belt )
   END_RUNG
   RUNG wire#powerrail
      Contact( #DI_Button_Water_Fountain_Get_Exit_Rework_Conveyor_Belt )
      Coil( #DB_Button_Water_Fountain_Get_Exit_Rework_Conveyor_Belt )
   END_RUNG
   // the same network as SCL:
   #DB_Sensor_Water_Fountain_Geting_Exit_Rework_Conveyor_Belt := #DI_Sensor_Water_Fountain_Geting_Exit_Rework_Conveyor_Belt;
   #DB_Button_Water_Fountain_Get_Exit_Rework_Conveyor_Belt := #DI_Button_Water_Fountain_Get_Exit_Rework_Conveyor_Belt;
END_REGION

REGION Network 4
   RUNG wire#powerrail
      Contact( #DI_Trigger_Read_Serial_Number_Exit_Functional_Test )
      Coil( #DB_Trigger_Read_Serial_Number_Exit_Functional_Test )
   END_RUNG
   RUNG wire#powerrail
      Contact( #DI_Sensor_Water_Fountain_Exit_Functional_Test_Spinner_Conveyor_Belt )
      Coil( #DB_Sensor_Water_Fountain_Exit_Functional_Test_Spinner_Conveyor_Belt )
   END_RUNG
   RUNG wire#powerrail
      Contact( #DI_Sensor_Water_Fountain_Exit_Functional_Test_After_Spinner_Conveyor_Belt )
      Coil( #DB_Sensor_Water_Fountain_Exit_Functional_Test_After_Spinner_Conveyor_Belt )
   END_RUNG
   // the same network as SCL:
   #DB_Trigger_Read_Serial_Number_Exit_Functional_Test := #DI_Trigger_Read_Serial_Number_Exit_Functional_Test;
   #DB_Sensor_Water_Fountain_Exit_Functional_Test_Spinner_Conveyor_Belt := #DI_Sensor_Water_Fountain_Exit_Functional_Test_Spinner_Conveyor_Belt;
   #DB_Sensor_Water_Fountain_Exit_Functional_Test_After_Spinner_Conveyor_Belt := #DI_Sensor_Water_Fountain_Exit_Functional_Test_After_Spinner_Conveyor_Belt;
END_REGION

REGION Network 5
   RUNG wire#powerrail
      Contact( #DI_Sensor_Water_Fountain_Geting_Entrace_Rework_Conveyor_Belt_Start )
      Coil( #DB_Sensor_Water_Fountain_Geting_Entrace_Rework_Conveyor_Belt_Start )
   END_RUNG
   RUNG wire#powerrail
      Contact( #DI_Sensor_Water_Fountain_Geting_Entrace_Rework_Conveyor_Belt_Finish )
      Coil( #DB_Sensor_Water_Fountain_Geting_Entrace_Rework_Conveyor_Belt_Finish )
   END_RUNG
   // the same network as SCL:
   #DB_Sensor_Water_Fountain_Geting_Entrace_Rework_Conveyor_Belt_Start := #DI_Sensor_Water_Fountain_Geting_Entrace_Rework_Conveyor_Belt_Start;
   #DB_Sensor_Water_Fountain_Geting_Entrace_Rework_Conveyor_Belt_Finish := #DI_Sensor_Water_Fountain_Geting_Entrace_Rework_Conveyor_Belt_Finish;
END_REGION

REGION Network 6
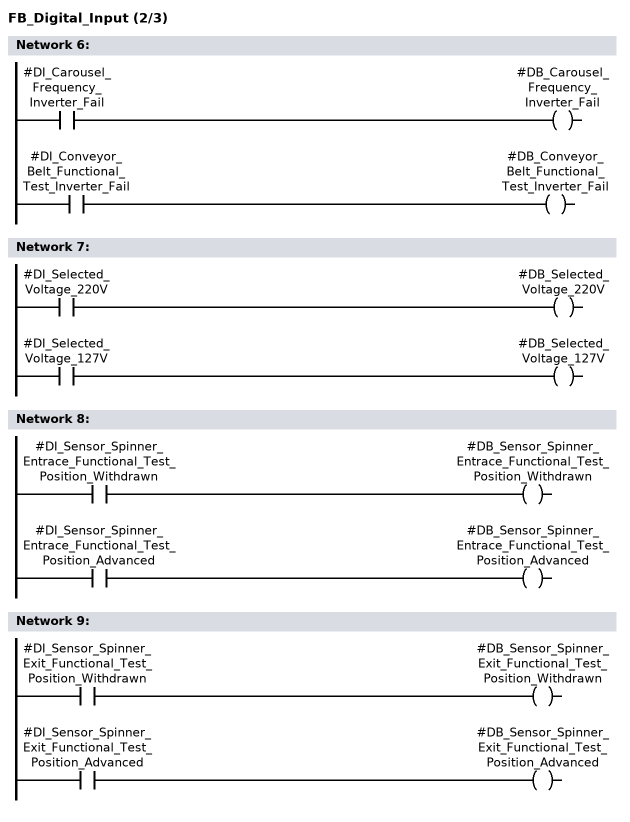
   RUNG wire#powerrail
      Contact( #DI_Carousel_Frequency_Inverter_Fail )
      Coil( #DB_Carousel_Frequency_Inverter_Fail )
   END_RUNG
   RUNG wire#powerrail
      Contact( #DI_Conveyor_Belt_Functional_Test_Inverter_Fail )
      Coil( #DB_Conveyor_Belt_Functional_Test_Inverter_Fail )
   END_RUNG
   // the same network as SCL:
   #DB_Carousel_Frequency_Inverter_Fail := #DI_Carousel_Frequency_Inverter_Fail;
   #DB_Conveyor_Belt_Functional_Test_Inverter_Fail := #DI_Conveyor_Belt_Functional_Test_Inverter_Fail;
END_REGION

REGION Network 7
   RUNG wire#powerrail
      Contact( #DI_Selected_Voltage_220V )
      Coil( #DB_Selected_Voltage_220V )
   END_RUNG
   RUNG wire#powerrail
      Contact( #DI_Selected_Voltage_127V )
      Coil( #DB_Selected_Voltage_127V )
   END_RUNG
   // the same network as SCL:
   #DB_Selected_Voltage_220V := #DI_Selected_Voltage_220V;
   #DB_Selected_Voltage_127V := #DI_Selected_Voltage_127V;
END_REGION

REGION Network 8
   RUNG wire#powerrail
      Contact( #DI_Sensor_Spinner_Entrace_Functional_Test_Position_Withdrawn )
      Coil( #DB_Sensor_Spinner_Entrace_Functional_Test_Position_Withdrawn )
   END_RUNG
   RUNG wire#powerrail
      Contact( #DI_Sensor_Spinner_Entrace_Functional_Test_Position_Advanced )
      Coil( #DB_Sensor_Spinner_Entrace_Functional_Test_Position_Advanced )
   END_RUNG
   // the same network as SCL:
   #DB_Sensor_Spinner_Entrace_Functional_Test_Position_Withdrawn := #DI_Sensor_Spinner_Entrace_Functional_Test_Position_Withdrawn;
   #DB_Sensor_Spinner_Entrace_Functional_Test_Position_Advanced := #DI_Sensor_Spinner_Entrace_Functional_Test_Position_Advanced;
END_REGION

REGION Network 9
   RUNG wire#powerrail
      Contact( #DI_Sensor_Spinner_Exit_Functional_Test_Position_Withdrawn )
      Coil( #DB_Sensor_Spinner_Exit_Functional_Test_Position_Withdrawn )
   END_RUNG
   RUNG wire#powerrail
      Contact( #DI_Sensor_Spinner_Exit_Functional_Test_Position_Advanced )
      Coil( #DB_Sensor_Spinner_Exit_Functional_Test_Position_Advanced )
   END_RUNG
   // the same network as SCL:
   #DB_Sensor_Spinner_Exit_Functional_Test_Position_Withdrawn := #DI_Sensor_Spinner_Exit_Functional_Test_Position_Withdrawn;
   #DB_Sensor_Spinner_Exit_Functional_Test_Position_Advanced := #DI_Sensor_Spinner_Exit_Functional_Test_Position_Advanced;
END_REGION

REGION Network 10
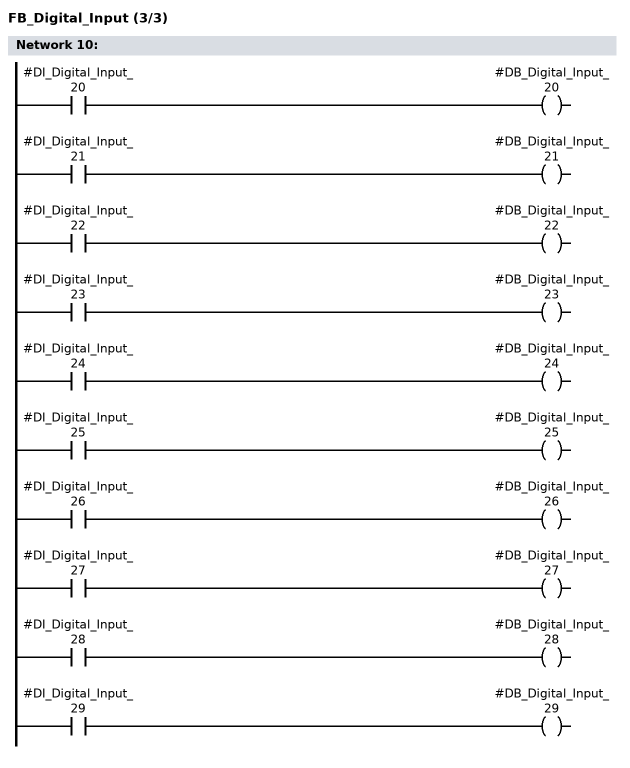
   RUNG wire#powerrail
      Contact( #DI_Digital_Input_20 )
      Coil( #DB_Digital_Input_20 )
   END_RUNG
   RUNG wire#powerrail
      Contact( #DI_Digital_Input_21 )
      Coil( #DB_Digital_Input_21 )
   END_RUNG
   RUNG wire#powerrail
      Contact( #DI_Digital_Input_22 )
      Coil( #DB_Digital_Input_22 )
   END_RUNG
   RUNG wire#powerrail
      Contact( #DI_Digital_Input_23 )
      Coil( #DB_Digital_Input_23 )
   END_RUNG
   RUNG wire#powerrail
      Contact( #DI_Digital_Input_24 )
      Coil( #DB_Digital_Input_24 )
   END_RUNG
   RUNG wire#powerrail
      Contact( #DI_Digital_Input_25 )
      Coil( #DB_Digital_Input_25 )
   END_RUNG
   RUNG wire#powerrail
      Contact( #DI_Digital_Input_26 )
      Coil( #DB_Digital_Input_26 )
   END_RUNG
   RUNG wire#powerrail
      Contact( #DI_Digital_Input_27 )
      Coil( #DB_Digital_Input_27 )
   END_RUNG
   RUNG wire#powerrail
      Contact( #DI_Digital_Input_28 )
      Coil( #DB_Digital_Input_28 )
   END_RUNG
   RUNG wire#powerrail
      Contact( #DI_Digital_Input_29 )
      Coil( #DB_Digital_Input_29 )
   END_RUNG
   // the same network as SCL:
   #DB_Digital_Input_20 := #DI_Digital_Input_20;
   #DB_Digital_Input_21 := #DI_Digital_Input_21;
   #DB_Digital_Input_22 := #DI_Digital_Input_22;
   #DB_Digital_Input_23 := #DI_Digital_Input_23;
   #DB_Digital_Input_24 := #DI_Digital_Input_24;
   #DB_Digital_Input_25 := #DI_Digital_Input_25;
   #DB_Digital_Input_26 := #DI_Digital_Input_26;
   #DB_Digital_Input_27 := #DI_Digital_Input_27;
   #DB_Digital_Input_28 := #DI_Digital_Input_28;
   #DB_Digital_Input_29 := #DI_Digital_Input_29;
END_REGION
END_FUNCTION_BLOCK

FUNCTION_BLOCK "FB_Analogic_Input"   // FB2, LAD
{ S7_Optimized_Access := 'TRUE' }
// Leitura das 2 Entradas Analogica de um CLP S7 1200 1214 DC/DC/DC
// stored: AutoNumber false, IsIECCheckEnabled true, MemoryReserve 100, SetENOAutomatically false
   VAR_INPUT
      Analogic_Input_0 { ExternalAccessible := 'False'; ExternalVisible := 'False'; ExternalWritable := 'False'} : Int;
      Analogic_Input_1 { ExternalAccessible := 'False'; ExternalVisible := 'False'; ExternalWritable := 'False'} : Int;
      Min_NormX_AI_0 { ExternalAccessible := 'False'; ExternalVisible := 'False'; ExternalWritable := 'False'} : Int := 0;
      Max_NormX_AI_0 { ExternalAccessible := 'False'; ExternalVisible := 'False'; ExternalWritable := 'False'} : Int := 27648;
      Min_NormX_AI_1 { ExternalAccessible := 'False'; ExternalVisible := 'False'; ExternalWritable := 'False'} : Int := 0;
      Max_NormX_AI_1 { ExternalAccessible := 'False'; ExternalVisible := 'False'; ExternalWritable := 'False'} : Int := 27648;
      Scale_Min_AI_0 { ExternalAccessible := 'False'; ExternalVisible := 'False'; ExternalWritable := 'False'} : Real;
      Scale_Max_AI_0 { ExternalAccessible := 'False'; ExternalVisible := 'False'; ExternalWritable := 'False'} : Real;
      Scale_Min_AI_1 { ExternalAccessible := 'False'; ExternalVisible := 'False'; ExternalWritable := 'False'} : Real;
      Scale_Max_AI_1 { ExternalAccessible := 'False'; ExternalVisible := 'False'; ExternalWritable := 'False'} : Real;
   END_VAR
   VAR_OUTPUT
      Value_Real_AI_0 { ExternalAccessible := 'False'; ExternalVisible := 'False'; ExternalWritable := 'False'} : Real;
      Value_Real_AI_1 { ExternalAccessible := 'False'; ExternalVisible := 'False'; ExternalWritable := 'False'} : Real;
      Value_UInt_AI_0 : UInt;
      Value_UInt_AI_1 : UInt;
   END_VAR
   VAR
      Norm_X_Out_AI_0 { ExternalAccessible := 'False'; ExternalVisible := 'False'; ExternalWritable := 'False'} : Real;
      Norm_X_Out_AI_1 { ExternalAccessible := 'False'; ExternalVisible := 'False'; ExternalWritable := 'False'} : Real;
   END_VAR
BEGIN

REGION Network 1: Analogic Input 0
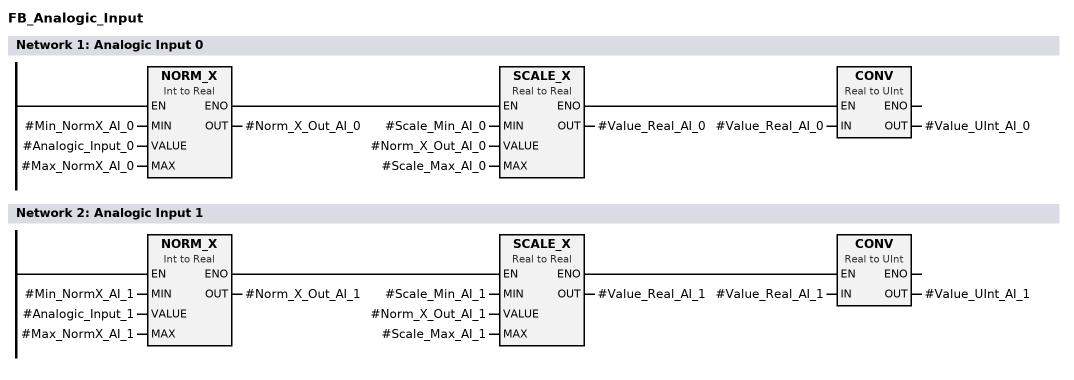
   RUNG wire#powerrail
      { S7_Templates := "[SrcType := Int, DestType := Real]" } Normalize(min := #Min_NormX_AI_0, value := #Analogic_Input_0, max := #Max_NormX_AI_0, out => #Norm_X_Out_AI_0)
      { S7_Templates := "[SrcType := Real, DestType := Real]" } Scale(min := #Scale_Min_AI_0, value := #Norm_X_Out_AI_0, max := #Scale_Max_AI_0, out => #Value_Real_AI_0)
      { S7_Templates := "[SrcType := Real, DestType := UInt]" } Convert(in := #Value_Real_AI_0, out => #Value_UInt_AI_0)
   END_RUNG
   // the same network as SCL:
   #Norm_X_Out_AI_0 := NORM_X(MIN := #Min_NormX_AI_0, VALUE := #Analogic_Input_0, MAX := #Max_NormX_AI_0);
   #Value_Real_AI_0 := SCALE_X(MIN := #Scale_Min_AI_0, VALUE := #Norm_X_Out_AI_0, MAX := #Scale_Max_AI_0);
   #Value_UInt_AI_0 := REAL_TO_UINT(#Value_Real_AI_0);
END_REGION

REGION Network 2: Analogic Input 1
   RUNG wire#powerrail
      { S7_Templates := "[SrcType := Int, DestType := Real]" } Normalize(min := #Min_NormX_AI_1, value := #Analogic_Input_1, max := #Max_NormX_AI_1, out => #Norm_X_Out_AI_1)
      { S7_Templates := "[SrcType := Real, DestType := Real]" } Scale(min := #Scale_Min_AI_1, value := #Norm_X_Out_AI_1, max := #Scale_Max_AI_1, out => #Value_Real_AI_1)
      { S7_Templates := "[SrcType := Real, DestType := UInt]" } Convert(in := #Value_Real_AI_1, out => #Value_UInt_AI_1)
   END_RUNG
   // the same network as SCL:
   #Norm_X_Out_AI_1 := NORM_X(MIN := #Min_NormX_AI_1, VALUE := #Analogic_Input_1, MAX := #Max_NormX_AI_1);
   #Value_Real_AI_1 := SCALE_X(MIN := #Scale_Min_AI_1, VALUE := #Norm_X_Out_AI_1, MAX := #Scale_Max_AI_1);
   #Value_UInt_AI_1 := REAL_TO_UINT(#Value_Real_AI_1);
END_REGION
END_FUNCTION_BLOCK

FUNCTION_BLOCK "FB_Digital_Output"   // FB3, LAD
{ S7_Optimized_Access := 'TRUE' }
// stored: AutoNumber false, MemoryReserve 100, SetENOAutomatically false
   VAR_INPUT
      DB_In_Emergency_Stop_Release : Bool;
      DB_In_Selected_Voltage_220V : Bool;
      DB_In_Selected_Voltage_127V : Bool;
      DB_Spin_Carousel_Frequency_Inverter_Speed_1 : Bool;
      DB_Spin_Carousel_Frequency_Inverter_Speed_2 : Bool;
      DB_Spin_Carousel_Frequency_Inverter_Speed_3 : Bool;
      DB_Conveyor_Belt_Frequency_Inverter_Speed_1 : Bool;
      DB_Conveyor_Belt_Frequency_Inverter_Speed_2 : Bool;
      DB_Conveyor_Belt_Frequency_Inverter_Speed_3 : Bool;
      DB_Turn_On_Conveyor_Belt_Motor_Spinner_Get_Entrace_Function_Test : Bool;
      DB_Turn_On_Conveyor_Belt_Motor_Rework_Conveyor_Belt_Get_Entrace_Functional_Test : Bool;
      DB_Turn_On_Conveyor_Belt_Motor_Spinner_Get_Exit_Functional_Test : Bool;
      DB_Turn_On_Conveyor_Belt_Motor_Rework_Conveyor_Belt_Get_Exit_Funcional_Test : Bool;
      DB_Open_Air_Pressure : Bool;
      DB_Valve_Advance_Spinner_Get_Entrace_Functional_Test : Bool;
      DB_Valve_Advance_Spinner_Get_Exit_Functional_Test : Bool;
      DB_Signal_Pre_Functional_Test_Production_Line : Bool;
      DB_Digital_Output_14 : Bool;
      DB_Digital_Output_15 : Bool;
      DB_Digital_Output_16 : Bool;
      DB_Digital_Output_17 : Bool;
      DB_Digital_Output_18 : Bool;
      DB_Digital_Output_19 : Bool;
      DB_Digital_Output_20 : Bool;
      DB_Digital_Output_21 : Bool;
      DB_Digital_Output_22 : Bool;
      DB_Digital_Output_23 : Bool;
      DB_Voltage_220V_Selected : Bool;
      DB_Voltage_127V_Selected : Bool;
   END_VAR
   VAR_OUTPUT
      DO_Spin_Carousel_Frequency_Inverter_Speed_1 : Bool;
      DO_Spin_Carousel_Frequency_Inverter_Speed_2 : Bool;
      DO_Spin_Carousel_Frequency_Inverter_Speed_3 : Bool;
      DO_Conveyor_Belt_Frequency_Inverter_Speed_1 : Bool;
      DO_Conveyor_Belt_Frequency_Inverter_Speed_2 : Bool;
      DO_Conveyor_Belt_Frequency_Inverter_Speed_3 : Bool;
      DO_Turn_On_Conveyor_Belt_Motor_Spinner_Get_Entrace_Function_Test : Bool;
      DO_Turn_On_Conveyor_Belt_Motor_Rework_Conveyor_Belt_Get_Entrace_Functional_Test : Bool;
      DO_Turn_On_Conveyor_Belt_Motor_Spinner_Get_Exit_Functional_Test : Bool;
      DO_Turn_On_Conveyor_Belt_Motor_Rework_Conveyor_Belt_Get_Exit_Funcional_Test : Bool;
      DO_Open_Air_Pressure : Bool;
      DO_Valve_Advance_Spinner_Entrace_Functional_Test : Bool;
      DO_Valve_Advance_Spinner_Exit_Functional_Test : Bool;
      DO_Signal_Pre_Functional_Test_Production_Line : Bool;
      DO_Digital_Output_14 : Bool;
      DO_Digital_Output_15 : Bool;
      DO_Digital_Output_16 : Bool;
      DO_Digital_Output_17 : Bool;
      DO_Digital_Output_18 : Bool;
      DO_Digital_Output_19 : Bool;
      DO_Digital_Output_20 : Bool;
      DO_Digital_Output_21 : Bool;
      DO_Digital_Output_22 : Bool;
      DO_Digital_Output_23 : Bool;
      DO_Voltage_220V_Selected : Bool;
      DO_Voltage_127V_Selected : Bool;
   END_VAR
   VAR
      Timer_Delay_Turn_On_220_V { S7_SetPoint := 'True'} : TON_TIME;
      Timer_Delay_Turn_On_127_V { S7_SetPoint := 'True'} : TON_TIME;
   END_VAR
BEGIN

REGION Network 1
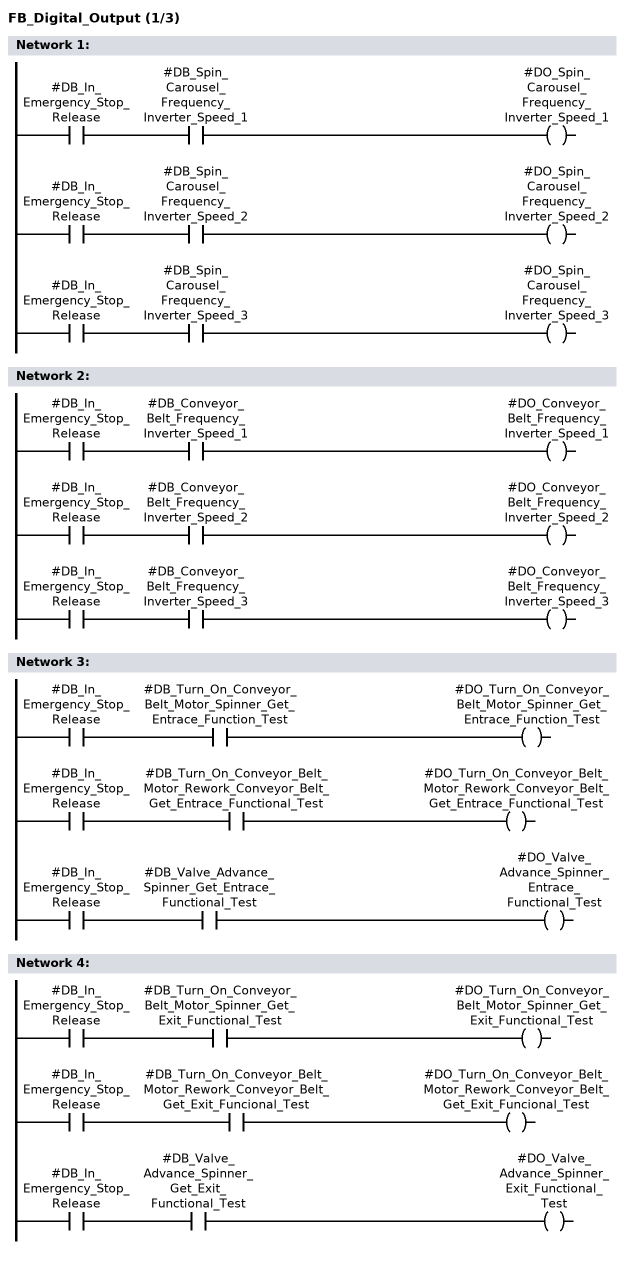
   RUNG wire#powerrail
      Contact( #DB_In_Emergency_Stop_Release )
      Contact( #DB_Spin_Carousel_Frequency_Inverter_Speed_1 )
      Coil( #DO_Spin_Carousel_Frequency_Inverter_Speed_1 )
   END_RUNG
   RUNG wire#powerrail
      Contact( #DB_In_Emergency_Stop_Release )
      Contact( #DB_Spin_Carousel_Frequency_Inverter_Speed_2 )
      Coil( #DO_Spin_Carousel_Frequency_Inverter_Speed_2 )
   END_RUNG
   RUNG wire#powerrail
      Contact( #DB_In_Emergency_Stop_Release )
      Contact( #DB_Spin_Carousel_Frequency_Inverter_Speed_3 )
      Coil( #DO_Spin_Carousel_Frequency_Inverter_Speed_3 )
   END_RUNG
   // the same network as SCL:
   #DO_Spin_Carousel_Frequency_Inverter_Speed_1 := #DB_In_Emergency_Stop_Release AND #DB_Spin_Carousel_Frequency_Inverter_Speed_1;
   #DO_Spin_Carousel_Frequency_Inverter_Speed_2 := #DB_In_Emergency_Stop_Release AND #DB_Spin_Carousel_Frequency_Inverter_Speed_2;
   #DO_Spin_Carousel_Frequency_Inverter_Speed_3 := #DB_In_Emergency_Stop_Release AND #DB_Spin_Carousel_Frequency_Inverter_Speed_3;
END_REGION

REGION Network 2
   RUNG wire#powerrail
      Contact( #DB_In_Emergency_Stop_Release )
      Contact( #DB_Conveyor_Belt_Frequency_Inverter_Speed_1 )
      Coil( #DO_Conveyor_Belt_Frequency_Inverter_Speed_1 )
   END_RUNG
   RUNG wire#powerrail
      Contact( #DB_In_Emergency_Stop_Release )
      Contact( #DB_Conveyor_Belt_Frequency_Inverter_Speed_2 )
      Coil( #DO_Conveyor_Belt_Frequency_Inverter_Speed_2 )
   END_RUNG
   RUNG wire#powerrail
      Contact( #DB_In_Emergency_Stop_Release )
      Contact( #DB_Conveyor_Belt_Frequency_Inverter_Speed_3 )
      Coil( #DO_Conveyor_Belt_Frequency_Inverter_Speed_3 )
   END_RUNG
   // the same network as SCL:
   #DO_Conveyor_Belt_Frequency_Inverter_Speed_1 := #DB_In_Emergency_Stop_Release AND #DB_Conveyor_Belt_Frequency_Inverter_Speed_1;
   #DO_Conveyor_Belt_Frequency_Inverter_Speed_2 := #DB_In_Emergency_Stop_Release AND #DB_Conveyor_Belt_Frequency_Inverter_Speed_2;
   #DO_Conveyor_Belt_Frequency_Inverter_Speed_3 := #DB_In_Emergency_Stop_Release AND #DB_Conveyor_Belt_Frequency_Inverter_Speed_3;
END_REGION

REGION Network 3
   RUNG wire#powerrail
      Contact( #DB_In_Emergency_Stop_Release )
      Contact( #DB_Turn_On_Conveyor_Belt_Motor_Spinner_Get_Entrace_Function_Test )
      Coil( #DO_Turn_On_Conveyor_Belt_Motor_Spinner_Get_Entrace_Function_Test )
   END_RUNG
   RUNG wire#powerrail
      Contact( #DB_In_Emergency_Stop_Release )
      Contact( #DB_Turn_On_Conveyor_Belt_Motor_Rework_Conveyor_Belt_Get_Entrace_Functional_Test )
      Coil( #DO_Turn_On_Conveyor_Belt_Motor_Rework_Conveyor_Belt_Get_Entrace_Functional_Test )
   END_RUNG
   RUNG wire#powerrail
      Contact( #DB_In_Emergency_Stop_Release )
      Contact( #DB_Valve_Advance_Spinner_Get_Entrace_Functional_Test )
      Coil( #DO_Valve_Advance_Spinner_Entrace_Functional_Test )
   END_RUNG
   // the same network as SCL:
   #DO_Turn_On_Conveyor_Belt_Motor_Spinner_Get_Entrace_Function_Test := #DB_In_Emergency_Stop_Release AND #DB_Turn_On_Conveyor_Belt_Motor_Spinner_Get_Entrace_Function_Test;
   #DO_Turn_On_Conveyor_Belt_Motor_Rework_Conveyor_Belt_Get_Entrace_Functional_Test := #DB_In_Emergency_Stop_Release AND #DB_Turn_On_Conveyor_Belt_Motor_Rework_Conveyor_Belt_Get_Entrace_Functional_Test;
   #DO_Valve_Advance_Spinner_Entrace_Functional_Test := #DB_In_Emergency_Stop_Release AND #DB_Valve_Advance_Spinner_Get_Entrace_Functional_Test;
END_REGION

REGION Network 4
   RUNG wire#powerrail
      Contact( #DB_In_Emergency_Stop_Release )
      Contact( #DB_Turn_On_Conveyor_Belt_Motor_Spinner_Get_Exit_Functional_Test )
      Coil( #DO_Turn_On_Conveyor_Belt_Motor_Spinner_Get_Exit_Functional_Test )
   END_RUNG
   RUNG wire#powerrail
      Contact( #DB_In_Emergency_Stop_Release )
      Contact( #DB_Turn_On_Conveyor_Belt_Motor_Rework_Conveyor_Belt_Get_Exit_Funcional_Test )
      Coil( #DO_Turn_On_Conveyor_Belt_Motor_Rework_Conveyor_Belt_Get_Exit_Funcional_Test )
   END_RUNG
   RUNG wire#powerrail
      Contact( #DB_In_Emergency_Stop_Release )
      Contact( #DB_Valve_Advance_Spinner_Get_Exit_Functional_Test )
      Coil( #DO_Valve_Advance_Spinner_Exit_Functional_Test )
   END_RUNG
   // the same network as SCL:
   #DO_Turn_On_Conveyor_Belt_Motor_Spinner_Get_Exit_Functional_Test := #DB_In_Emergency_Stop_Release AND #DB_Turn_On_Conveyor_Belt_Motor_Spinner_Get_Exit_Functional_Test;
   #DO_Turn_On_Conveyor_Belt_Motor_Rework_Conveyor_Belt_Get_Exit_Funcional_Test := #DB_In_Emergency_Stop_Release AND #DB_Turn_On_Conveyor_Belt_Motor_Rework_Conveyor_Belt_Get_Exit_Funcional_Test;
   #DO_Valve_Advance_Spinner_Exit_Functional_Test := #DB_In_Emergency_Stop_Release AND #DB_Valve_Advance_Spinner_Get_Exit_Functional_Test;
END_REGION

REGION Network 5
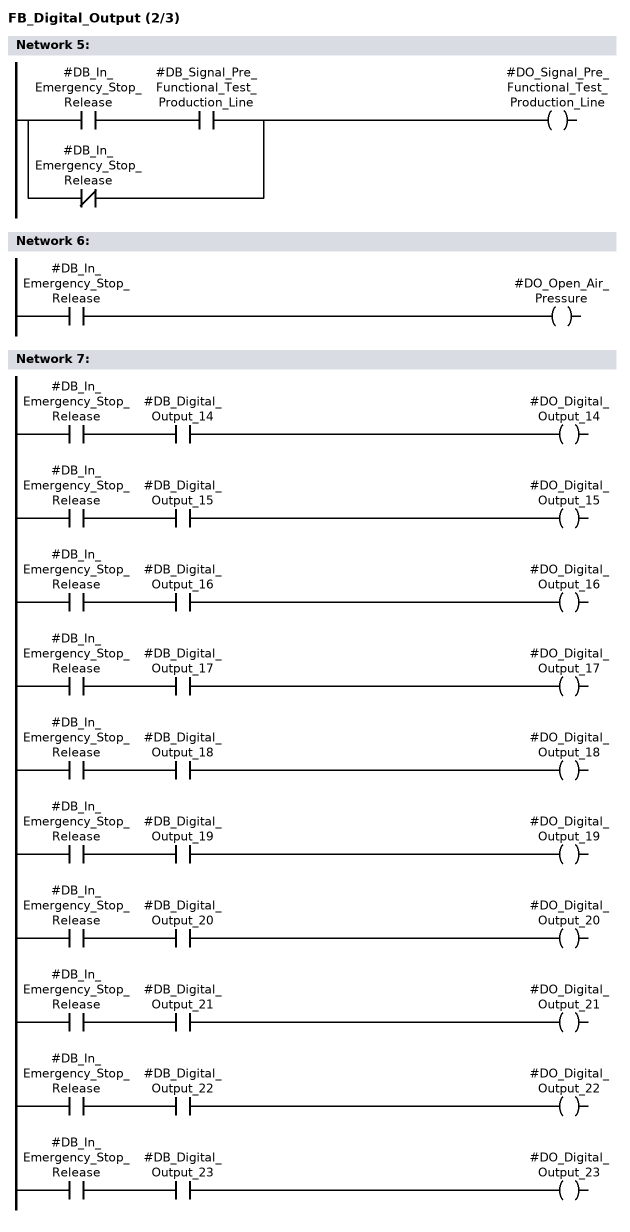
   RUNG wire#powerrail
      Contact( #DB_In_Emergency_Stop_Release )
      Contact( #DB_Signal_Pre_Functional_Test_Production_Line )
      wire#w1
      Coil( #DO_Signal_Pre_Functional_Test_Production_Line )
   END_RUNG
   RUNG wire#powerrail
      I_Contact( #DB_In_Emergency_Stop_Release )
   END_RUNG wire#w1
   // the same network as SCL:
   #DO_Signal_Pre_Functional_Test_Production_Line := (#DB_In_Emergency_Stop_Release AND #DB_Signal_Pre_Functional_Test_Production_Line) OR NOT #DB_In_Emergency_Stop_Release;
END_REGION

REGION Network 6
   RUNG wire#powerrail
      Contact( #DB_In_Emergency_Stop_Release )
      Coil( #DO_Open_Air_Pressure )
   END_RUNG
   // the same network as SCL:
   #DO_Open_Air_Pressure := #DB_In_Emergency_Stop_Release;
END_REGION

REGION Network 7
   RUNG wire#powerrail
      Contact( #DB_In_Emergency_Stop_Release )
      Contact( #DB_Digital_Output_14 )
      Coil( #DO_Digital_Output_14 )
   END_RUNG
   RUNG wire#powerrail
      Contact( #DB_In_Emergency_Stop_Release )
      Contact( #DB_Digital_Output_15 )
      Coil( #DO_Digital_Output_15 )
   END_RUNG
   RUNG wire#powerrail
      Contact( #DB_In_Emergency_Stop_Release )
      Contact( #DB_Digital_Output_16 )
      Coil( #DO_Digital_Output_16 )
   END_RUNG
   RUNG wire#powerrail
      Contact( #DB_In_Emergency_Stop_Release )
      Contact( #DB_Digital_Output_17 )
      Coil( #DO_Digital_Output_17 )
   END_RUNG
   RUNG wire#powerrail
      Contact( #DB_In_Emergency_Stop_Release )
      Contact( #DB_Digital_Output_18 )
      Coil( #DO_Digital_Output_18 )
   END_RUNG
   RUNG wire#powerrail
      Contact( #DB_In_Emergency_Stop_Release )
      Contact( #DB_Digital_Output_19 )
      Coil( #DO_Digital_Output_19 )
   END_RUNG
   RUNG wire#powerrail
      Contact( #DB_In_Emergency_Stop_Release )
      Contact( #DB_Digital_Output_20 )
      Coil( #DO_Digital_Output_20 )
   END_RUNG
   RUNG wire#powerrail
      Contact( #DB_In_Emergency_Stop_Release )
      Contact( #DB_Digital_Output_21 )
      Coil( #DO_Digital_Output_21 )
   END_RUNG
   RUNG wire#powerrail
      Contact( #DB_In_Emergency_Stop_Release )
      Contact( #DB_Digital_Output_22 )
      Coil( #DO_Digital_Output_22 )
   END_RUNG
   RUNG wire#powerrail
      Contact( #DB_In_Emergency_Stop_Release )
      Contact( #DB_Digital_Output_23 )
      Coil( #DO_Digital_Output_23 )
   END_RUNG
   // the same network as SCL:
   #DO_Digital_Output_14 := #DB_In_Emergency_Stop_Release AND #DB_Digital_Output_14;
   #DO_Digital_Output_15 := #DB_In_Emergency_Stop_Release AND #DB_Digital_Output_15;
   #DO_Digital_Output_16 := #DB_In_Emergency_Stop_Release AND #DB_Digital_Output_16;
   #DO_Digital_Output_17 := #DB_In_Emergency_Stop_Release AND #DB_Digital_Output_17;
   #DO_Digital_Output_18 := #DB_In_Emergency_Stop_Release AND #DB_Digital_Output_18;
   #DO_Digital_Output_19 := #DB_In_Emergency_Stop_Release AND #DB_Digital_Output_19;
   #DO_Digital_Output_20 := #DB_In_Emergency_Stop_Release AND #DB_Digital_Output_20;
   #DO_Digital_Output_21 := #DB_In_Emergency_Stop_Release AND #DB_Digital_Output_21;
   #DO_Digital_Output_22 := #DB_In_Emergency_Stop_Release AND #DB_Digital_Output_22;
   #DO_Digital_Output_23 := #DB_In_Emergency_Stop_Release AND #DB_Digital_Output_23;
END_REGION

REGION Network 8
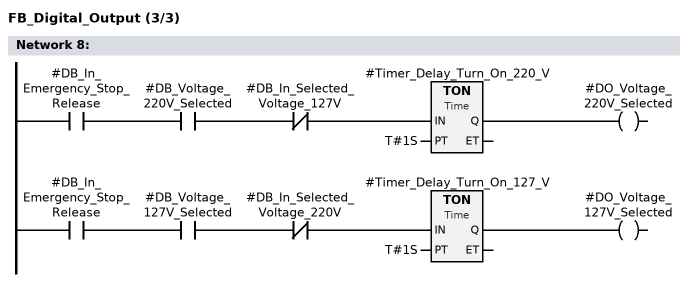
   RUNG wire#powerrail
      Contact( #DB_In_Emergency_Stop_Release )
      Contact( #DB_Voltage_220V_Selected )
      I_Contact( #DB_In_Selected_Voltage_127V )
      { S7_Templates := "time_type := Time" } #Timer_Delay_Turn_On_220_V.TON(pt := T#1S, et =>)
      Coil( #DO_Voltage_220V_Selected )
   END_RUNG
   RUNG wire#powerrail
      Contact( #DB_In_Emergency_Stop_Release )
      Contact( #DB_Voltage_127V_Selected )
      I_Contact( #DB_In_Selected_Voltage_220V )
      { S7_Templates := "time_type := Time" } #Timer_Delay_Turn_On_127_V.TON(pt := T#1S, et =>)
      Coil( #DO_Voltage_127V_Selected )
   END_RUNG
   // the same network as SCL:
   #Timer_Delay_Turn_On_220_V(IN := #DB_In_Emergency_Stop_Release AND #DB_Voltage_220V_Selected AND NOT #DB_In_Selected_Voltage_127V,   // TON
                           PT := T#1S);
   #DO_Voltage_220V_Selected := #Timer_Delay_Turn_On_220_V.Q;
   #Timer_Delay_Turn_On_127_V(IN := #DB_In_Emergency_Stop_Release AND #DB_Voltage_127V_Selected AND NOT #DB_In_Selected_Voltage_220V,   // TON
                           PT := T#1S);
   #DO_Voltage_127V_Selected := #Timer_Delay_Turn_On_127_V.Q;
END_REGION
END_FUNCTION_BLOCK

FUNCTION_BLOCK "FB_IO_Device"   // FB4, LAD
{ S7_Optimized_Access := 'TRUE' }
// stored: MemoryReserve 100, SetENOAutomatically false
   VAR_INPUT
      Life_Trigger : Bool;
      Emergency_Stop_Release : Bool;
      Trigger_Read_Serial_Number_Entrace_Functional_Test : Bool;
      Trigger_Read_Serial_Number_Exit_Functional_Test : Bool;
      Selected_Voltage_220V : Bool;
      Selected_Voltage_127V : Bool;
      Carousel_Frequency_Inverter_Fail : Bool;
      Conveyor_Belt_Functional_Test_Inverter_Fail : Bool;
      In : "IO_Device_Inputs";
   END_VAR
   VAR_OUTPUT
      Start : Bool;
      Manual_Turn_On_Motor_Caroussel : Bool;
      Manual_Turn_On_Motor_Conveyor_Belt : Bool;
      Water_Foutain_Fail_Functional_Test : Bool;
      Select_Motor_Speed : SInt;
      Carousel_Voltage_Selection : SInt;
      Out : "IO_Device_Outputs";
   END_VAR
BEGIN

REGION Network 1
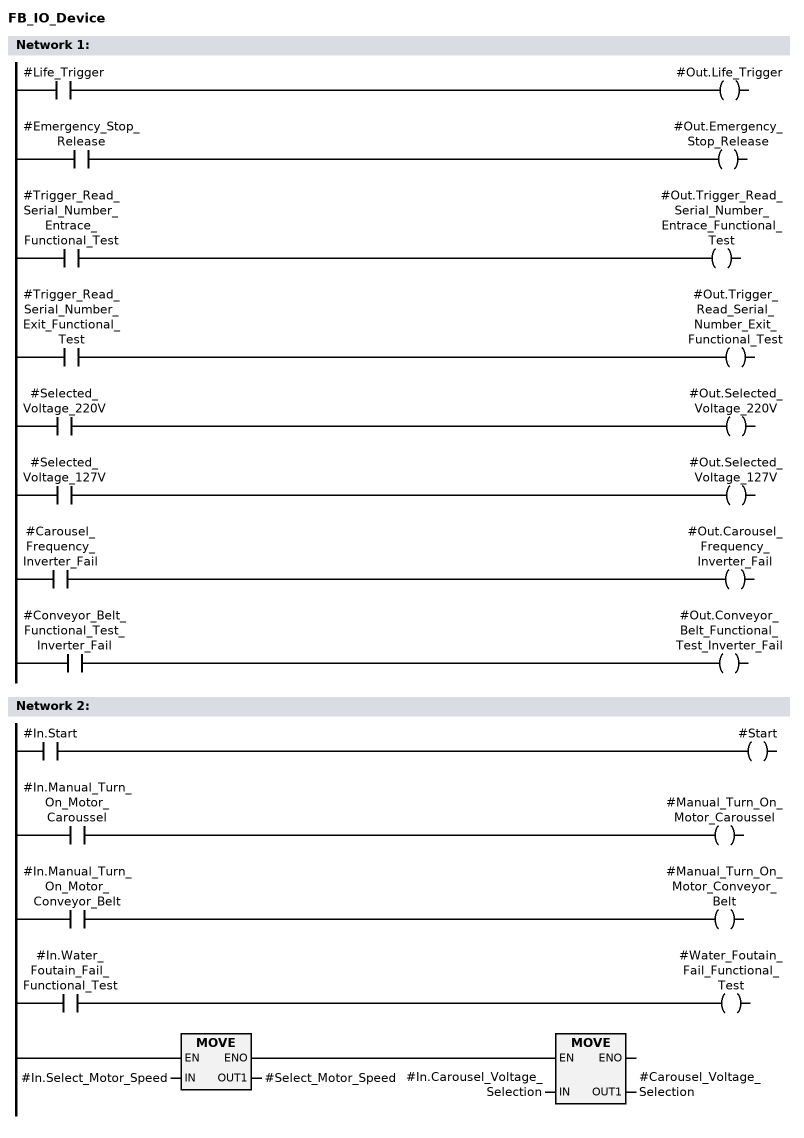
   RUNG wire#powerrail
      Contact( #Life_Trigger )
      Coil( #Out.Life_Trigger )
   END_RUNG
   RUNG wire#powerrail
      Contact( #Emergency_Stop_Release )
      Coil( #Out.Emergency_Stop_Release )
   END_RUNG
   RUNG wire#powerrail
      Contact( #Trigger_Read_Serial_Number_Entrace_Functional_Test )
      Coil( #Out.Trigger_Read_Serial_Number_Entrace_Functional_Test )
   END_RUNG
   RUNG wire#powerrail
      Contact( #Trigger_Read_Serial_Number_Exit_Functional_Test )
      Coil( #Out.Trigger_Read_Serial_Number_Exit_Functional_Test )
   END_RUNG
   RUNG wire#powerrail
      Contact( #Selected_Voltage_220V )
      Coil( #Out.Selected_Voltage_220V )
   END_RUNG
   RUNG wire#powerrail
      Contact( #Selected_Voltage_127V )
      Coil( #Out.Selected_Voltage_127V )
   END_RUNG
   RUNG wire#powerrail
      Contact( #Carousel_Frequency_Inverter_Fail )
      Coil( #Out.Carousel_Frequency_Inverter_Fail )
   END_RUNG
   RUNG wire#powerrail
      Contact( #Conveyor_Belt_Functional_Test_Inverter_Fail )
      Coil( #Out.Conveyor_Belt_Functional_Test_Inverter_Fail )
   END_RUNG
   // the same network as SCL:
   #Out.Life_Trigger := #Life_Trigger;
   #Out.Emergency_Stop_Release := #Emergency_Stop_Release;
   #Out.Trigger_Read_Serial_Number_Entrace_Functional_Test := #Trigger_Read_Serial_Number_Entrace_Functional_Test;
   #Out.Trigger_Read_Serial_Number_Exit_Functional_Test := #Trigger_Read_Serial_Number_Exit_Functional_Test;
   #Out.Selected_Voltage_220V := #Selected_Voltage_220V;
   #Out.Selected_Voltage_127V := #Selected_Voltage_127V;
   #Out.Carousel_Frequency_Inverter_Fail := #Carousel_Frequency_Inverter_Fail;
   #Out.Conveyor_Belt_Functional_Test_Inverter_Fail := #Conveyor_Belt_Functional_Test_Inverter_Fail;
END_REGION

REGION Network 2
   RUNG wire#powerrail
      Contact( #In.Start )
      Coil( #Start )
   END_RUNG
   RUNG wire#powerrail
      Contact( #In.Manual_Turn_On_Motor_Caroussel )
      Coil( #Manual_Turn_On_Motor_Caroussel )
   END_RUNG
   RUNG wire#powerrail
      Contact( #In.Manual_Turn_On_Motor_Conveyor_Belt )
      Coil( #Manual_Turn_On_Motor_Conveyor_Belt )
   END_RUNG
   RUNG wire#powerrail
      Contact( #In.Water_Foutain_Fail_Functional_Test )
      Coil( #Water_Foutain_Fail_Functional_Test )
   END_RUNG
   RUNG wire#powerrail
      Move(in := #In.Select_Motor_Speed, out1 => #Select_Motor_Speed)
      Move(in := #In.Carousel_Voltage_Selection, out1 => #Carousel_Voltage_Selection)
   END_RUNG
   // the same network as SCL:
   #Start := #In.Start;
   #Manual_Turn_On_Motor_Caroussel := #In.Manual_Turn_On_Motor_Caroussel;
   #Manual_Turn_On_Motor_Conveyor_Belt := #In.Manual_Turn_On_Motor_Conveyor_Belt;
   #Water_Foutain_Fail_Functional_Test := #In.Water_Foutain_Fail_Functional_Test;
   #Select_Motor_Speed := #In.Select_Motor_Speed;
   #Carousel_Voltage_Selection := #In.Carousel_Voltage_Selection;
END_REGION
END_FUNCTION_BLOCK

FUNCTION_BLOCK "FB_Recive_Water_Fountain_From_Rework"   // FB5, LAD
{ S7_Optimized_Access := 'TRUE' }
// stored: MemoryReserve 100, SetENOAutomatically false
   VAR_INPUT
      Emergency_Stop_Release : Bool;
      Start : Bool;
      Sensor_Water_Fountain_Before_Entrace_Functional_Test_Spinner_Conveyor_Belt : Bool;
      Sensor_Water_Fountain_Entrace_Functional_Test_Spinner_Conveyor_Belt : Bool;
      Sensor_Spinner_Entrace_Functional_Test_Position_Withdrawn : Bool;
      Sensor_Spinner_Entrace_Functional_Test_Position_Advanced : Bool;
      Sensor_Water_Fountain_Entrace_Functional_Test_After_Spinner_Conveyor_Belt : Bool;
      Sensor_Water_Fountain_Geting_Exit_Rework_Conveyor_Belt : Bool;
      Button_Water_Fountain_Get_Exit_Rework_Conveyor_Belt : Bool;
      Trigger_Read_Serial_Number_Entrace_Functional_Test : Bool;
   END_VAR
   VAR_OUTPUT
      Turn_On_Conveyor_Belt_Motor_Spinner_Get_Entrace_Function_Test : Bool;
      Valve_Advance_Spinner_Entrace_Functional_Test : Bool;
      Signal_Pre_Functional_Test_Production_Line : Bool;
   END_VAR
   VAR
      Aux_Trig_0 : Bool;
      Aux_Trig_1 : Bool;
      Aux_Trig_2 : Bool;
      Aux_Trig_3 : Bool;
      Aux_Trig_4 : Bool;
      Aux_Trig_5 : Bool;
      Aux_Trig_6 : Bool;
      Aux_Trig_7 : Bool;
      Aux_Trig_8 : Bool;
      Aux_Trig_9 : Bool;
      Button_Rework_Pressed : Bool;
      "Counter" : USInt;
      Timer_Delay_Turn_On_Motor_Spinner_Conveyor_Belt : TON_TIME;
      Counter_Water_Fountain_Entrace_Functional_Test { S7_SetPoint := 'True'} : CTUD_USINT;
   END_VAR
   VAR RETAIN
      Timer_Delay_Spin_Advanced { S7_SetPoint := 'True'} : TON_TIME;
   END_VAR
   VAR
      Timer_Delay_Spin_Withdrawn { S7_SetPoint := 'True'} : TON_TIME;
   END_VAR
   VAR_TEMP   // added for the SCL form of the ladder/FBD networks
      _w1 : Bool;
      _w2 : Bool;
   END_VAR
BEGIN

REGION Network 1
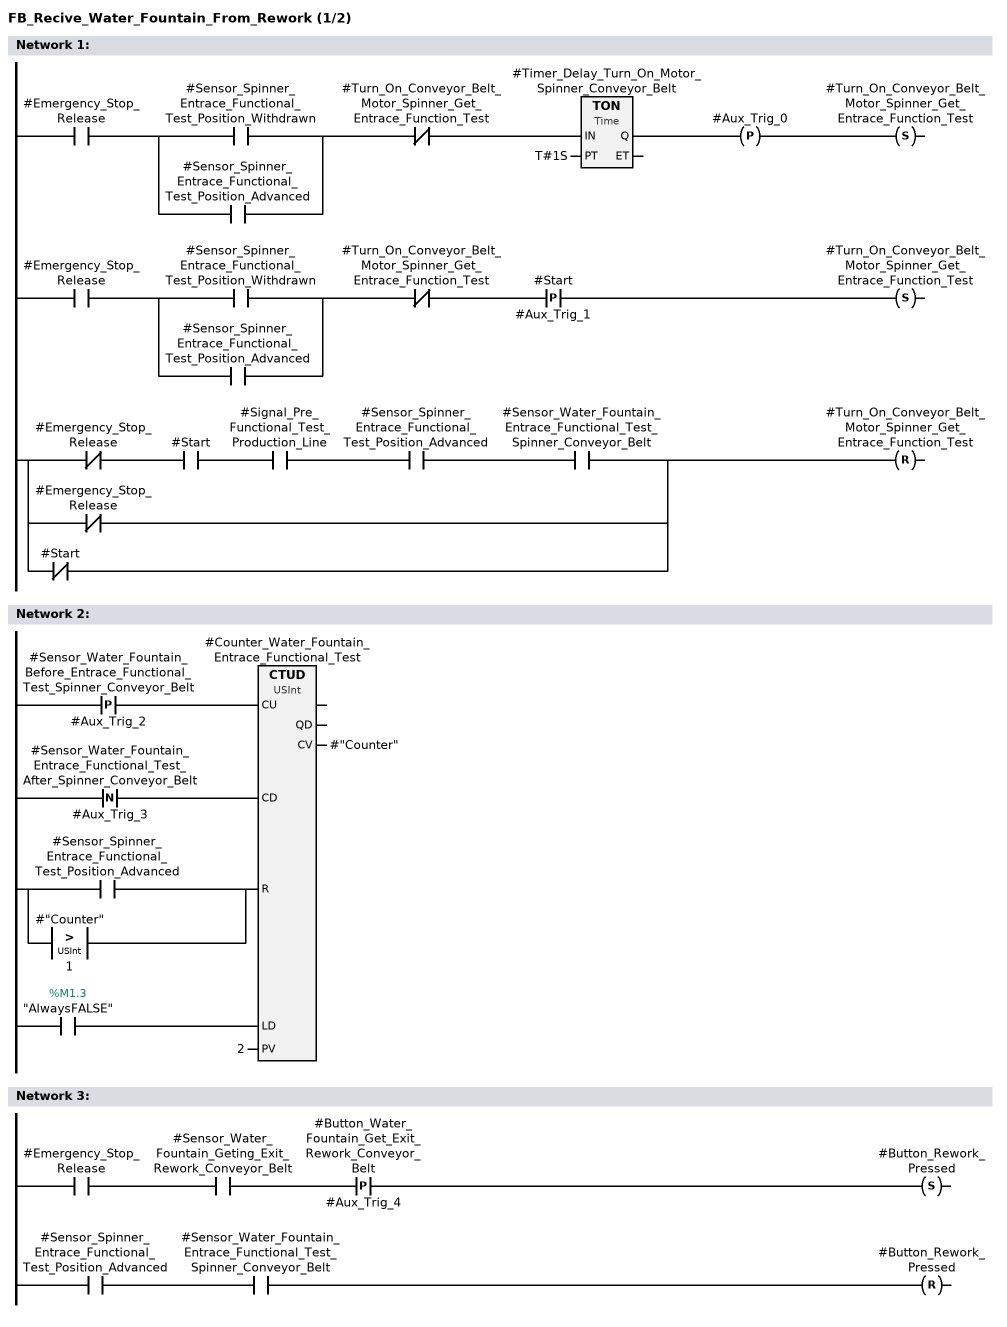
   RUNG wire#powerrail
      Contact( #Emergency_Stop_Release )
      wire#w1
      Contact( #Sensor_Spinner_Entrace_Functional_Test_Position_Withdrawn )
      wire#w2
      I_Contact( #Turn_On_Conveyor_Belt_Motor_Spinner_Get_Entrace_Function_Test )
      { S7_Templates := "time_type := Time" } #Timer_Delay_Turn_On_Motor_Spinner_Conveyor_Belt.TON(pt := T#1S, et =>)
      P_Trig( #Aux_Trig_0 )
      S_Coil( #Turn_On_Conveyor_Belt_Motor_Spinner_Get_Entrace_Function_Test )
   END_RUNG
   RUNG wire#w1
      Contact( #Sensor_Spinner_Entrace_Functional_Test_Position_Advanced )
   END_RUNG wire#w2
   RUNG wire#powerrail
      Contact( #Emergency_Stop_Release )
      wire#w3
      Contact( #Sensor_Spinner_Entrace_Functional_Test_Position_Withdrawn )
      wire#w4
      I_Contact( #Turn_On_Conveyor_Belt_Motor_Spinner_Get_Entrace_Function_Test )
      P_Contact(operand := #Start, bit := #Aux_Trig_1)
      S_Coil( #Turn_On_Conveyor_Belt_Motor_Spinner_Get_Entrace_Function_Test )
   END_RUNG
   RUNG wire#w3
      Contact( #Sensor_Spinner_Entrace_Functional_Test_Position_Advanced )
   END_RUNG wire#w4
   RUNG wire#powerrail
      I_Contact( #Emergency_Stop_Release )
      Contact( #Start )
      Contact( #Signal_Pre_Functional_Test_Production_Line )
      Contact( #Sensor_Spinner_Entrace_Functional_Test_Position_Advanced )
      Contact( #Sensor_Water_Fountain_Entrace_Functional_Test_Spinner_Conveyor_Belt )
      wire#w5
      R_Coil( #Turn_On_Conveyor_Belt_Motor_Spinner_Get_Entrace_Function_Test )
   END_RUNG
   RUNG wire#powerrail
      I_Contact( #Emergency_Stop_Release )
   END_RUNG wire#w5
   RUNG wire#powerrail
      I_Contact( #Start )
   END_RUNG wire#w5
   // the same network as SCL:
   #Timer_Delay_Turn_On_Motor_Spinner_Conveyor_Belt(IN := #Emergency_Stop_Release AND (#Sensor_Spinner_Entrace_Functional_Test_Position_Withdrawn OR #Sensor_Spinner_Entrace_Functional_Test_Position_Advanced) AND NOT #Turn_On_Conveyor_Belt_Motor_Spinner_Get_Entrace_Function_Test,   // TON
                           PT := T#1S);
   #_w1 := #Timer_Delay_Turn_On_Motor_Spinner_Conveyor_Belt.Q AND NOT #Aux_Trig_0;   // rising edge
   #Aux_Trig_0 := #Timer_Delay_Turn_On_Motor_Spinner_Conveyor_Belt.Q;
   IF #_w1 THEN #Turn_On_Conveyor_Belt_Motor_Spinner_Get_Entrace_Function_Test := TRUE; END_IF;
   #_w2 := #Emergency_Stop_Release AND (#Sensor_Spinner_Entrace_Functional_Test_Position_Withdrawn OR #Sensor_Spinner_Entrace_Functional_Test_Position_Advanced) AND NOT #Turn_On_Conveyor_Belt_Motor_Spinner_Get_Entrace_Function_Test AND #Start AND NOT #Aux_Trig_1;   // rising edge of #Start
   #Aux_Trig_1 := #Start;
   IF #_w2 THEN #Turn_On_Conveyor_Belt_Motor_Spinner_Get_Entrace_Function_Test := TRUE; END_IF;
   IF (NOT #Emergency_Stop_Release AND #Start AND #Signal_Pre_Functional_Test_Production_Line AND #Sensor_Spinner_Entrace_Functional_Test_Position_Advanced AND #Sensor_Water_Fountain_Entrace_Functional_Test_Spinner_Conveyor_Belt) OR NOT #Emergency_Stop_Release OR NOT #Start THEN
       #Turn_On_Conveyor_Belt_Motor_Spinner_Get_Entrace_Function_Test := FALSE;
   END_IF;
END_REGION

REGION Network 2
   RUNG wire#powerrail
      P_Contact(operand := #Sensor_Water_Fountain_Before_Entrace_Functional_Test_Spinner_Conveyor_Belt, bit := #Aux_Trig_2)
      { S7_Templates := "value_type := USInt" } #Counter_Water_Fountain_Entrace_Functional_Test.CTUD(cd := wire#w1, r := wire#w2, ld := wire#w3, pv := 2, qd =>, cv => #"Counter")
   END_RUNG
   RUNG wire#powerrail
      N_Contact(operand := #Sensor_Water_Fountain_Entrace_Functional_Test_After_Spinner_Conveyor_Belt, bit := #Aux_Trig_3)
   END_RUNG wire#w1
   RUNG wire#powerrail
      Contact( #Sensor_Spinner_Entrace_Functional_Test_Position_Advanced )
   END_RUNG wire#w2
   RUNG wire#powerrail
      { S7_Templates := "SrcType := USInt" } GT_Contact(in1 := #"Counter", in2 := 1)
   END_RUNG wire#w2
   RUNG wire#powerrail
      Contact( "AlwaysFALSE" )
   END_RUNG wire#w3
   // the same network as SCL:
   #_w1 := #Sensor_Water_Fountain_Before_Entrace_Functional_Test_Spinner_Conveyor_Belt AND NOT #Aux_Trig_2;   // rising edge of #Sensor_Water_Fountain_Before_Entrace_Functional_Test_Spinner_Conveyor_Belt
   #Aux_Trig_2 := #Sensor_Water_Fountain_Before_Entrace_Functional_Test_Spinner_Conveyor_Belt;
   #_w2 := NOT #Sensor_Water_Fountain_Entrace_Functional_Test_After_Spinner_Conveyor_Belt AND #Aux_Trig_3;   // falling edge of #Sensor_Water_Fountain_Entrace_Functional_Test_After_Spinner_Conveyor_Belt
   #Aux_Trig_3 := #Sensor_Water_Fountain_Entrace_Functional_Test_After_Spinner_Conveyor_Belt;
   #Counter_Water_Fountain_Entrace_Functional_Test(CU := #_w1,   // CTUD
                           CD := #_w2,
                           R := #Sensor_Spinner_Entrace_Functional_Test_Position_Advanced OR (#"Counter" > 1),
                           LD := "AlwaysFALSE",
                           PV := 2,
                           CV => #"Counter");
END_REGION

REGION Network 3
   RUNG wire#powerrail
      Contact( #Emergency_Stop_Release )
      Contact( #Sensor_Water_Fountain_Geting_Exit_Rework_Conveyor_Belt )
      P_Contact(operand := #Button_Water_Fountain_Get_Exit_Rework_Conveyor_Belt, bit := #Aux_Trig_4)
      S_Coil( #Button_Rework_Pressed )
   END_RUNG
   RUNG wire#powerrail
      Contact( #Sensor_Spinner_Entrace_Functional_Test_Position_Advanced )
      Contact( #Sensor_Water_Fountain_Entrace_Functional_Test_Spinner_Conveyor_Belt )
      R_Coil( #Button_Rework_Pressed )
   END_RUNG
   // the same network as SCL:
   #_w1 := #Emergency_Stop_Release AND #Sensor_Water_Fountain_Geting_Exit_Rework_Conveyor_Belt AND #Button_Water_Fountain_Get_Exit_Rework_Conveyor_Belt AND NOT #Aux_Trig_4;   // rising edge of #Button_Water_Fountain_Get_Exit_Rework_Conveyor_Belt
   #Aux_Trig_4 := #Button_Water_Fountain_Get_Exit_Rework_Conveyor_Belt;
   IF #_w1 THEN #Button_Rework_Pressed := TRUE; END_IF;
   IF #Sensor_Spinner_Entrace_Functional_Test_Position_Advanced AND #Sensor_Water_Fountain_Entrace_Functional_Test_Spinner_Conveyor_Belt THEN
       #Button_Rework_Pressed := FALSE;
   END_IF;
END_REGION

REGION Network 4
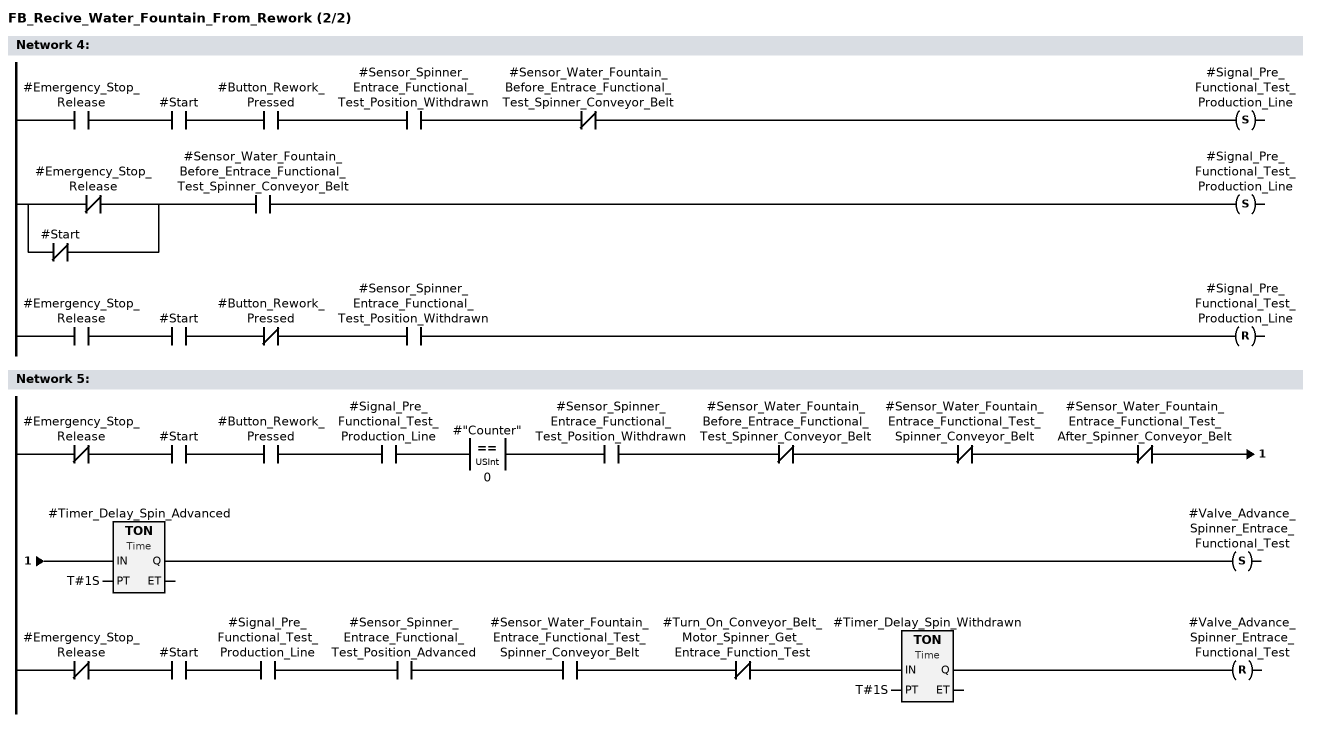
   RUNG wire#powerrail
      Contact( #Emergency_Stop_Release )
      Contact( #Start )
      Contact( #Button_Rework_Pressed )
      Contact( #Sensor_Spinner_Entrace_Functional_Test_Position_Withdrawn )
      I_Contact( #Sensor_Water_Fountain_Before_Entrace_Functional_Test_Spinner_Conveyor_Belt )
      S_Coil( #Signal_Pre_Functional_Test_Production_Line )
   END_RUNG
   RUNG wire#powerrail
      I_Contact( #Emergency_Stop_Release )
      wire#w1
      Contact( #Sensor_Water_Fountain_Before_Entrace_Functional_Test_Spinner_Conveyor_Belt )
      S_Coil( #Signal_Pre_Functional_Test_Production_Line )
   END_RUNG
   RUNG wire#powerrail
      I_Contact( #Start )
   END_RUNG wire#w1
   RUNG wire#powerrail
      Contact( #Emergency_Stop_Release )
      Contact( #Start )
      I_Contact( #Button_Rework_Pressed )
      Contact( #Sensor_Spinner_Entrace_Functional_Test_Position_Withdrawn )
      R_Coil( #Signal_Pre_Functional_Test_Production_Line )
   END_RUNG
   // the same network as SCL:
   IF #Emergency_Stop_Release AND #Start AND #Button_Rework_Pressed AND #Sensor_Spinner_Entrace_Functional_Test_Position_Withdrawn AND NOT #Sensor_Water_Fountain_Before_Entrace_Functional_Test_Spinner_Conveyor_Belt THEN
       #Signal_Pre_Functional_Test_Production_Line := TRUE;
   END_IF;
   IF (NOT #Emergency_Stop_Release OR NOT #Start) AND #Sensor_Water_Fountain_Before_Entrace_Functional_Test_Spinner_Conveyor_Belt THEN
       #Signal_Pre_Functional_Test_Production_Line := TRUE;
   END_IF;
   IF #Emergency_Stop_Release AND #Start AND NOT #Button_Rework_Pressed AND #Sensor_Spinner_Entrace_Functional_Test_Position_Withdrawn THEN
       #Signal_Pre_Functional_Test_Production_Line := FALSE;
   END_IF;
END_REGION

REGION Network 5
   RUNG wire#powerrail
      I_Contact( #Emergency_Stop_Release )
      Contact( #Start )
      Contact( #Button_Rework_Pressed )
      Contact( #Signal_Pre_Functional_Test_Production_Line )
      { S7_Templates := "SrcType := USInt" } EQ_Contact(in1 := #"Counter", in2 := 0)
      Contact( #Sensor_Spinner_Entrace_Functional_Test_Position_Withdrawn )
      I_Contact( #Sensor_Water_Fountain_Before_Entrace_Functional_Test_Spinner_Conveyor_Belt )
      I_Contact( #Sensor_Water_Fountain_Entrace_Functional_Test_Spinner_Conveyor_Belt )
      I_Contact( #Sensor_Water_Fountain_Entrace_Functional_Test_After_Spinner_Conveyor_Belt )
      { S7_Templates := "time_type := Time" } #Timer_Delay_Spin_Advanced.TON(pt := T#1S, et =>)
      S_Coil( #Valve_Advance_Spinner_Entrace_Functional_Test )
   END_RUNG
   RUNG wire#powerrail
      I_Contact( #Emergency_Stop_Release )
      Contact( #Start )
      Contact( #Signal_Pre_Functional_Test_Production_Line )
      Contact( #Sensor_Spinner_Entrace_Functional_Test_Position_Advanced )
      Contact( #Sensor_Water_Fountain_Entrace_Functional_Test_Spinner_Conveyor_Belt )
      I_Contact( #Turn_On_Conveyor_Belt_Motor_Spinner_Get_Entrace_Function_Test )
      { S7_Templates := "time_type := Time" } #Timer_Delay_Spin_Withdrawn.TON(pt := T#1S, et =>)
      R_Coil( #Valve_Advance_Spinner_Entrace_Functional_Test )
   END_RUNG
   // the same network as SCL:
   #Timer_Delay_Spin_Advanced(IN := NOT #Emergency_Stop_Release AND #Start AND #Button_Rework_Pressed AND #Signal_Pre_Functional_Test_Production_Line AND (#"Counter" = 0) AND #Sensor_Spinner_Entrace_Functional_Test_Position_Withdrawn AND NOT #Sensor_Water_Fountain_Before_Entrace_Functional_Test_Spinner_Conveyor_Belt AND NOT #Sensor_Water_Fountain_Entrace_Functional_Test_Spinner_Conveyor_Belt AND NOT #Sensor_Water_Fountain_Entrace_Functional_Test_After_Spinner_Conveyor_Belt,   // TON
                           PT := T#1S);
   IF #Timer_Delay_Spin_Advanced.Q THEN #Valve_Advance_Spinner_Entrace_Functional_Test := TRUE; END_IF;
   #Timer_Delay_Spin_Withdrawn(IN := NOT #Emergency_Stop_Release AND #Start AND #Signal_Pre_Functional_Test_Production_Line AND #Sensor_Spinner_Entrace_Functional_Test_Position_Advanced AND #Sensor_Water_Fountain_Entrace_Functional_Test_Spinner_Conveyor_Belt AND NOT #Turn_On_Conveyor_Belt_Motor_Spinner_Get_Entrace_Function_Test,   // TON
                           PT := T#1S);
   IF #Timer_Delay_Spin_Withdrawn.Q THEN #Valve_Advance_Spinner_Entrace_Functional_Test := FALSE; END_IF;
END_REGION
END_FUNCTION_BLOCK

